LIN {X 0,Y 420.675,Z 239.811,A -85,B 0,C 180,E1 -10145.839,E2 -10145.839} C_VEL
LIN {X 0,Y 420.884,Z 242.407,A -85,B 0,C 180,E1 -10146.375,E2 -10146.375} C_VEL
LIN {X 0,Y 419.869,Z 259.45,A -85,B 0,C 180,E1 -10149.746,E2 -10149.746} C_VEL
LIN {X 0,Y 419.418,Z 267.017,A -85,B 0,C 180,E1 -10151.23,E2 -10151.23} C_VEL
LIN {X 0,Y 423.148,Z 292.501,A -85,B 0,C 180,E1 -10151.829,E2 -10151.829} C_VEL
LIN {X 0,Y 422.342,Z 375.452,A -85,B 0,C 180,E1 -10153.256,E2 -10153.256} C_VEL
LIN {X 0,Y 421.795,Z 388.688,A -85,B 0,C 180,E1 -10153.67,E2 -10153.67} C_VEL
LIN {X 0,Y 421.223,Z 401.426,A -85,B 0,C 180,E1 -10154.269,E2 -10154.269} C_VEL
LIN {X 0,Y 420.604,Z 412.728,A -85,B 0,C 180,E1 -10154.99,E2 -10154.99} C_VEL
LIN {X 0,Y 419.83,Z 424.418,A -85,B 0,C 180,E1 -10155.953,E2 -10155.953} C_VEL
LIN {X 0,Y 419.241,Z 434.93,A -85,B 0,C 180,E1 -10157.043,E2 -10157.043} C_VEL
LIN {X 0,Y 418.677,Z 443.516,A -85,B 0,C 180,E1 -10158.134,E2 -10158.134} C_VEL
LIN {X 0,Y 418.09,Z 451.424,A -85,B 0,C 180,E1 -10159.344,E2 -10159.344} C_VEL
LIN {X 0,Y 417.649,Z 459.143,A -85,B 0,C 180,E1 -10160.801,E2 -10160.801} C_VEL
LIN {X 0,Y 417.351,Z 465.34,A -85,B 0,C 180,E1 -10162.258,E2 -10162.258} C_VEL
LIN {X 0,Y 417.171,Z 470.222,A -85,B 0,C 180,E1 -10163.702,E2 -10163.702} C_VEL
LIN {X 0,Y 417.106,Z 474.036,A -85,B 0,C 180,E1 -10165.167,E2 -10165.167} C_VEL
LIN {X 0,Y 417.014,Z 475.982,A -85,B 0,C 180,E1 -10166.135,E2 -10166.135} C_VEL
LIN {X 0,Y 417.029,Z 477.511,A -85,B 0,C 180,E1 -10167.102,E2 -10167.102} C_VEL
LIN {X 0,Y 417.056,Z 478.586,A -85,B 0,C 180,E1 -10168.069,E2 -10168.069} C_VEL
LIN {X 0,Y 417.005,Z 479.55,A -85,B 0,C 180,E1 -10170,E2 -10170} C_VEL
LIN {X 0,Y 417.011,Z 479.453,A -85,B 0,C 180,E1 -10170.966,E2 -10170.966} C_VEL
LIN {X 0,Y 417.056,Z 478.925,A -85,B 0,C 180,E1 -10171.931,E2 -10171.931} C_VEL
LIN {X 0,Y 417.026,Z 477.997,A -85,B 0,C 180,E1 -10172.898,E2 -10172.898} C_VEL
LIN {X 0,Y 417.106,Z 474.952,A -85,B 0,C 180,E1 -10174.833,E2 -10174.833} C_VEL
LIN {X 0,Y 417.141,Z 471.563,A -85,B 0,C 180,E1 -10176.261,E2 -10176.261} C_VEL
LIN {X 0,Y 417.395,Z 466.962,A -85,B 0,C 180,E1 -10177.741,E2 -10177.741} C_VEL
LIN {X 0,Y 417.821,Z 460.107,A -85,B 0,C 180,E1 -10179.439,E2 -10179.439} C_VEL
LIN {X 0,Y 418.342,Z 452.686,A -85,B 0,C 180,E1 -10180.894,E2 -10180.894} C_VEL
LIN {X 0,Y 419.064,Z 445.134,A -85,B 0,C 180,E1 -10182.101,E2 -10182.101} C_VEL
LIN {X 0,Y 419.775,Z 436.004,A -85,B 0,C 180,E1 -10183.309,E2 -10183.309} C_VEL
LIN {X 0,Y 420.395,Z 426.465,A -85,B 0,C 180,E1 -10184.343,E2 -10184.343} C_VEL
LIN {X 0,Y 421.316,Z 414.675,A -85,B 0,C 180,E1 -10185.356,E2 -10185.356} C_VEL
LIN {X 0,Y 421.992,Z 404.07,A -85,B 0,C 180,E1 -10186.074,E2 -10186.074} C_VEL
LIN {X 0,Y 422.721,Z 391.294,A -85,B 0,C 180,E1 -10186.728,E2 -10186.728} C_VEL
LIN {X 0,Y 423.278,Z 378.466,A -85,B 0,C 180,E1 -10187.172,E2 -10187.172} C_VEL
LIN {X 0,Y 423.711,Z 360.488,A -85,B 0,C 180,E1 -10187.524,E2 -10187.524} C_VEL
LIN {X 0,Y 424.326,Z 291.938,A -85,B 0,C 180,E1 -10188.705,E2 -10188.705} C_VEL
LIN {X 0,Y 420.251,Z 268.65,A -85,B 0,C 180,E1 -10189.331,E2 -10189.331} C_VEL
LIN {X 0,Y 419.936,Z 266.884,A -85,B 0,C 180,E1 -10189.38,E2 -10189.38} C_VEL
LIN {X 0,Y 421.141,Z 249.854,A -85,B 0,C 180,E1 -10192.791,E2 -10192.791} C_VEL
LIN {X 0,Y 421.47,Z 243.375,A -85,B 0,C 180,E1 -10194.113,E2 -10194.113} C_VEL
LIN {X 0,Y 419.295,Z 232.058,A -85,B 0,C 180,E1 -10196.639,E2 -10196.639} C_VEL
LIN {X 0,Y 418.289,Z 227.385,A -85,B 0,C 180,E1 -10197.747,E2 -10197.747} C_VEL
LIN {X 0,Y 418.24,Z 227.389,A -85,B 0,C 180,E1 -10201.019,E2 -10201.019} C_VEL
LIN {X 0,Y 418.25,Z 227.388,A -85,B 0,C 180,E1 -10203.677,E2 -10203.677} C_VEL
LIN {X 0,Y 418.24,Z 227.389,A -85,B 0,C 180,E1 -10207.224,E2 -10207.224} C_VEL
LIN {X 0,Y 418.244,Z 227.389,A -85,B 0,C 180,E1 -10209.683,E2 -10209.683} C_VEL
LIN {X 0,Y 418.224,Z 227.387,A -85,B 0,C 180,E1 -10212.32,E2 -10212.32} C_VEL
LIN {X 0,Y 418.236,Z 227.388,A -85,B 0,C 180,E1 -10215.109,E2 -10215.109} C_VEL
LIN {X 0,Y 418.235,Z 227.389,A -85,B 0,C 180,E1 -10217.766,E2 -10217.766} C_VEL
LIN {X 0,Y 418.238,Z 227.389,A -85,B 0,C 180,E1 -10221.557,E2 -10221.557} C_VEL
LIN {X 0,Y 418.258,Z 227.385,A -85,B 0,C 180,E1 -10225.159,E2 -10225.159} C_VEL
LIN {X 0,Y 418.246,Z 227.385,A -85,B 0,C 180,E1 -10227.472,E2 -10227.472} C_VEL
LIN {X 0,Y 418.265,Z 227.377,A -85,B 0,C 180,E1 -10230.897,E2 -10230.897} C_VEL
LIN {X 0,Y 418.238,Z 227.38,A -85,B 0,C 180,E1 -10234.094,E2 -10234.094} C_VEL
LIN {X 0,Y 418.232,Z 227.39,A -85,B 0,C 180,E1 -10237.264,E2 -10237.264} C_VEL
LIN {X 0,Y 418.284,Z 227.378,A -85,B 0,C 180,E1 -10240.364,E2 -10240.364} C_VEL
LIN {X 0,Y 418.317,Z 227.374,A -85,B 0,C 180,E1 -10243.405,E2 -10243.405} C_VEL
LIN {X 0,Y 418.347,Z 227.372,A -85,B 0,C 180,E1 -10246.999,E2 -10246.999} C_VEL
LIN {X 0,Y 418.341,Z 227.371,A -85,B 0,C 180,E1 -10250.329,E2 -10250.329} C_VEL
LIN {X 0,Y 418.494,Z 227.35,A -85,B 0,C 180,E1 -10253.249,E2 -10253.249} C_VEL
LIN {X 0,Y 418.333,Z 227.375,A -85,B 0,C 180,E1 -10255.182,E2 -10255.182} C_VEL
LIN {X 0,Y 418.54,Z 227.342,A -85,B 0,C 180,E1 -10258.076,E2 -10258.076} C_VEL
LIN {X 0,Y 418.67,Z 227.331,A -85,B 0,C 180,E1 -10260,E2 -10260} C_VEL
LIN {X 0,Y 418.494,Z 227.35,A -85,B 0,C 180,E1 -10262.888,E2 -10262.888} C_VEL
LIN {X 0,Y 418.46,Z 227.356,A -85,B 0,C 180,E1 -10266.487,E2 -10266.487} C_VEL
LIN {X 0,Y 418.339,Z 227.376,A -85,B 0,C 180,E1 -10269.672,E2 -10269.672} C_VEL
LIN {X 0,Y 418.348,Z 227.37,A -85,B 0,C 180,E1 -10273.001,E2 -10273.001} C_VEL
LIN {X 0,Y 418.313,Z 227.374,A -85,B 0,C 180,E1 -10276.735,E2 -10276.735} C_VEL
LIN {X 0,Y 418.271,Z 227.382,A -85,B 0,C 180,E1 -10279.79,E2 -10279.79} C_VEL
LIN {X 0,Y 418.238,Z 227.378,A -85,B 0,C 180,E1 -10282.736,E2 -10282.736} C_VEL
LIN {X 0,Y 418.262,Z 227.378,A -85,B 0,C 180,E1 -10285.905,E2 -10285.905} C_VEL
LIN {X 0,Y 418.27,Z 227.384,A -85,B 0,C 180,E1 -10289.105,E2 -10289.105} C_VEL
LIN {X 0,Y 418.259,Z 227.383,A -85,B 0,C 180,E1 -10292.844,E2 -10292.844} C_VEL
LIN {X 0,Y 418.245,Z 227.381,A -85,B 0,C 180,E1 -10296.238,E2 -10296.238} C_VEL
LIN {X 0,Y 418.245,Z 227.388,A -85,B 0,C 180,E1 -10299.683,E2 -10299.683} C_VEL
LIN {X 0,Y 418.225,Z 227.387,A -85,B 0,C 180,E1 -10302.32,E2 -10302.32} C_VEL
LIN {X 0,Y 418.237,Z 227.39,A -85,B 0,C 180,E1 -10305.109,E2 -10305.109} C_VEL
LIN {X 0,Y 418.236,Z 227.391,A -85,B 0,C 180,E1 -10307.766,E2 -10307.766} C_VEL
LIN {X 0,Y 418.24,Z 227.394,A -85,B 0,C 180,E1 -10311.557,E2 -10311.557} C_VEL
LIN {X 0,Y 418.26,Z 227.389,A -85,B 0,C 180,E1 -10315.159,E2 -10315.159} C_VEL
LIN {X 0,Y 418.248,Z 227.388,A -85,B 0,C 180,E1 -10317.472,E2 -10317.472} C_VEL
LIN {X 0,Y 418.294,Z 227.523,A -85,B 0,C 180,E1 -10320.496,E2 -10320.496} C_VEL
LIN {X 0,Y 420.231,Z 237.183,A -85,B 0,C 180,E1 -10322.823,E2 -10322.823} C_VEL
LIN {X 0,Y 420.452,Z 242.272,A -85,B 0,C 180,E1 -10323.974,E2 -10323.974} C_VEL
LIN {X 0,Y 420.296,Z 245.419,A -85,B 0,C 180,E1 -10324.663,E2 -10324.663} C_VEL
LIN {X 0,Y 424.472,Z 264.589,A -85,B 0,C 180,E1 -10325.245,E2 -10325.245} C_VEL
LIN {X 0,Y 424.757,Z 269.362,A -85,B 0,C 180,E1 -10325.345,E2 -10325.345} C_VEL
LIN {X 0,Y 423.574,Z 353.087,A -85,B 0,C 180,E1 -10326.792,E2 -10326.792} C_VEL
LIN {X 0,Y 423.157,Z 366.435,A -85,B 0,C 180,E1 -10327.22,E2 -10327.22} C_VEL
LIN {X 0,Y 422.58,Z 379.229,A -85,B 0,C 180,E1 -10327.832,E2 -10327.832} C_VEL
LIN {X 0,Y 421.894,Z 390.948,A -85,B 0,C 180,E1 -10328.598,E2 -10328.598} C_VEL
LIN {X 0,Y 421.084,Z 402.881,A -85,B 0,C 180,E1 -10329.61,E2 -10329.61} C_VEL
LIN {X 0,Y 420.227,Z 413.237,A -85,B 0,C 180,E1 -10330.713,E2 -10330.713} C_VEL
LIN {X 0,Y 419.492,Z 422.499,A -85,B 0,C 180,E1 -10331.944,E2 -10331.944} C_VEL
LIN {X 0,Y 418.921,Z 429.828,A -85,B 0,C 180,E1 -10333.125,E2 -10333.125} C_VEL
LIN {X 0,Y 418.261,Z 437.559,A -85,B 0,C 180,E1 -10334.654,E2 -10334.654} C_VEL
LIN {X 0,Y 417.805,Z 444.366,A -85,B 0,C 180,E1 -10336.379,E2 -10336.379} C_VEL
LIN {X 0,Y 417.464,Z 449.019,A -85,B 0,C 180,E1 -10337.927,E2 -10337.927} C_VEL
LIN {X 0,Y 417.198,Z 452.2,A -85,B 0,C 180,E1 -10339.321,E2 -10339.321} C_VEL
LIN {X 0,Y 417.05,Z 454.001,A -85,B 0,C 180,E1 -10340.402,E2 -10340.402} C_VEL
LIN {X 0,Y 416.349,Z 455.082,A -85,B 0,C 180,E1 -10341.198,E2 -10341.198} C_VEL
LIN {X 0,Y 413.478,Z 456.229,A -85,B 0,C 180,E1 -10342.5,E2 -10342.5} C_VEL
LIN {X 0,Y 411.07,Z 456.634,A -85,B 0,C 180,E1 -10343.556,E2 -10343.556} C_VEL
LIN {X 0,Y 410.033,Z 456.603,A -85,B 0,C 180,E1 -10344.372,E2 -10344.372} C_VEL
LIN {X 0,Y 409.946,Z 456.468,A -85,B 0,C 180,E1 -10344.649,E2 -10344.649} C_VEL
LIN {X 0,Y 409.913,Z 455.619,A -85,B 0,C 180,E1 -10346.068,E2 -10346.068} C_VEL
LIN {X 0,Y 409.974,Z 454.491,A -85,B 0,C 180,E1 -10347.052,E2 -10347.052} C_VEL
LIN {X 0,Y 410.055,Z 452.937,A -85,B 0,C 180,E1 -10348.036,E2 -10348.036} C_VEL
LIN {X 0,Y 410.166,Z 449.828,A -85,B 0,C 180,E1 -10349.509,E2 -10349.509} C_VEL
LIN {X 0,Y 410.32,Z 445.675,A -85,B 0,C 180,E1 -10350.981,E2 -10350.981} C_VEL
LIN {X 0,Y 410.761,Z 439.351,A -85,B 0,C 180,E1 -10352.697,E2 -10352.697} C_VEL
LIN {X 0,Y 411.135,Z 432.478,A -85,B 0,C 180,E1 -10354.166,E2 -10354.166} C_VEL
LIN {X 0,Y 411.87,Z 423.849,A -85,B 0,C 180,E1 -10355.631,E2 -10355.631} C_VEL
LIN {X 0,Y 412.563,Z 415.025,A -85,B 0,C 180,E1 -10356.848,E2 -10356.848} C_VEL
LIN {X 0,Y 413.211,Z 405.345,A -85,B 0,C 180,E1 -10357.943,E2 -10357.943} C_VEL
LIN {X 0,Y 413.883,Z 394.726,A -85,B 0,C 180,E1 -10358.914,E2 -10358.914} C_VEL
LIN {X 0,Y 414.541,Z 382.831,A -85,B 0,C 180,E1 -10359.761,E2 -10359.761} C_VEL
LIN {X 0,Y 415.116,Z 370.445,A -85,B 0,C 180,E1 -10360.425,E2 -10360.425} C_VEL
LIN {X 0,Y 415.446,Z 357.479,A -85,B 0,C 180,E1 -10360.912,E2 -10360.912} C_VEL
LIN {X 0,Y 415.769,Z 341.674,A -85,B 0,C 180,E1 -10361.246,E2 -10361.246} C_VEL
LIN {X 0,Y 416.563,Z 266.126,A -85,B 0,C 180,E1 -10362.546,E2 -10362.546} C_VEL
LIN {X 0,Y 412.835,Z 245.467,A -85,B 0,C 180,E1 -10363.099,E2 -10363.099} C_VEL
LIN {X 0,Y 413.033,Z 237.818,A -85,B 0,C 180,E1 -10364.787,E2 -10364.787} C_VEL
LIN {X 0,Y 411.275,Z 228.258,A -85,B 0,C 180,E1 -10367.055,E2 -10367.055} C_VEL
LIN {X 0,Y 411.234,Z 228.257,A -85,B 0,C 180,E1 -10369.987,E2 -10369.987} C_VEL
LIN {X 0,Y 411.199,Z 228.262,A -85,B 0,C 180,E1 -10373.148,E2 -10373.148} C_VEL
LIN {X 0,Y 411.206,Z 228.263,A -85,B 0,C 180,E1 -10376.383,E2 -10376.383} C_VEL
LIN {X 0,Y 411.2,Z 228.26,A -85,B 0,C 180,E1 -10379.713,E2 -10379.713} C_VEL
LIN {X 0,Y 411.209,Z 228.261,A -85,B 0,C 180,E1 -10383.156,E2 -10383.156} C_VEL
LIN {X 0,Y 411.194,Z 228.266,A -85,B 0,C 180,E1 -10386.552,E2 -10386.552} C_VEL
LIN {X 0,Y 411.213,Z 228.258,A -85,B 0,C 180,E1 -10389.727,E2 -10389.727} C_VEL
LIN {X 0,Y 411.175,Z 228.265,A -85,B 0,C 180,E1 -10393.133,E2 -10393.133} C_VEL
LIN {X 0,Y 411.169,Z 228.264,A -85,B 0,C 180,E1 -10395.881,E2 -10395.881} C_VEL
LIN {X 0,Y 411.162,Z 228.271,A -85,B 0,C 180,E1 -10398.772,E2 -10398.772} C_VEL
LIN {X 0,Y 411.193,Z 228.262,A -85,B 0,C 180,E1 -10402.026,E2 -10402.026} C_VEL
LIN {X 0,Y 411.207,Z 228.259,A -85,B 0,C 180,E1 -10405.666,E2 -10405.666} C_VEL
LIN {X 0,Y 411.191,Z 228.263,A -85,B 0,C 180,E1 -10409.152,E2 -10409.152} C_VEL
LIN {X 0,Y 411.259,Z 228.258,A -85,B 0,C 180,E1 -10412.522,E2 -10412.522} C_VEL
LIN {X 0,Y 411.218,Z 228.258,A -85,B 0,C 180,E1 -10415.784,E2 -10415.784} C_VEL
LIN {X 0,Y 411.197,Z 228.264,A -85,B 0,C 180,E1 -10418.966,E2 -10418.966} C_VEL
LIN {X 0,Y 411.246,Z 228.256,A -85,B 0,C 180,E1 -10422.084,E2 -10422.084} C_VEL
LIN {X 0,Y 411.259,Z 228.254,A -85,B 0,C 180,E1 -10425.147,E2 -10425.147} C_VEL
LIN {X 0,Y 411.284,Z 228.252,A -85,B 0,C 180,E1 -10428.167,E2 -10428.167} C_VEL
LIN {X 0,Y 411.319,Z 228.247,A -85,B 0,C 180,E1 -10431.154,E2 -10431.154} C_VEL
LIN {X 0,Y 411.444,Z 228.231,A -85,B 0,C 180,E1 -10434.117,E2 -10434.117} C_VEL
LIN {X 0,Y 411.512,Z 228.222,A -85,B 0,C 180,E1 -10438.042,E2 -10438.042} C_VEL
LIN {X 0,Y 411.639,Z 228.206,A -85,B 0,C 180,E1 -10440,E2 -10440} C_VEL
LIN {X 0,Y 411.45,Z 228.232,A -85,B 0,C 180,E1 -10442.937,E2 -10442.937} C_VEL
LIN {X 0,Y 411.461,Z 228.231,A -85,B 0,C 180,E1 -10446.867,E2 -10446.867} C_VEL
LIN {X 0,Y 411.354,Z 228.245,A -85,B 0,C 180,E1 -10448.845,E2 -10448.845} C_VEL
LIN {X 0,Y 411.284,Z 228.25,A -85,B 0,C 180,E1 -10451.833,E2 -10451.833} C_VEL
LIN {X 0,Y 411.261,Z 228.256,A -85,B 0,C 180,E1 -10454.853,E2 -10454.853} C_VEL
LIN {X 0,Y 411.246,Z 228.255,A -85,B 0,C 180,E1 -10457.915,E2 -10457.915} C_VEL
LIN {X 0,Y 411.197,Z 228.263,A -85,B 0,C 180,E1 -10461.034,E2 -10461.034} C_VEL
LIN {X 0,Y 411.212,Z 228.261,A -85,B 0,C 180,E1 -10464.216,E2 -10464.216} C_VEL
LIN {X 0,Y 411.19,Z 228.261,A -85,B 0,C 180,E1 -10467.483,E2 -10467.483} C_VEL
LIN {X 0,Y 411.189,Z 228.265,A -85,B 0,C 180,E1 -10470.848,E2 -10470.848} C_VEL
LIN {X 0,Y 411.205,Z 228.264,A -85,B 0,C 180,E1 -10474.334,E2 -10474.334} C_VEL
LIN {X 0,Y 411.186,Z 228.263,A -85,B 0,C 180,E1 -10477.975,E2 -10477.975} C_VEL
LIN {X 0,Y 411.158,Z 228.266,A -85,B 0,C 180,E1 -10481.227,E2 -10481.227} C_VEL
LIN {X 0,Y 411.176,Z 228.27,A -85,B 0,C 180,E1 -10484.491,E2 -10484.491} C_VEL
LIN {X 0,Y 411.173,Z 228.266,A -85,B 0,C 180,E1 -10488.194,E2 -10488.194} C_VEL
LIN {X 0,Y 411.211,Z 228.263,A -85,B 0,C 180,E1 -10490.775,E2 -10490.775} C_VEL
LIN {X 0,Y 411.198,Z 228.267,A -85,B 0,C 180,E1 -10494.471,E2 -10494.471} C_VEL
LIN {X 0,Y 411.208,Z 228.262,A -85,B 0,C 180,E1 -10496.873,E2 -10496.873} C_VEL
LIN {X 0,Y 411.234,Z 228.262,A -85,B 0,C 180,E1 -10500.644,E2 -10500.644} C_VEL
LIN {X 0,Y 411.267,Z 228.273,A -85,B 0,C 180,E1 -10502.938,E2 -10502.938} C_VEL
LIN {X 0,Y 413.851,Z 242.011,A -85,B 0,C 180,E1 -10505.948,E2 -10505.948} C_VEL
LIN {X 0,Y 413.184,Z 254.87,A -85,B 0,C 180,E1 -10508.549,E2 -10508.549} C_VEL
LIN {X 0,Y 412.444,Z 266.837,A -85,B 0,C 180,E1 -10510.94,E2 -10510.94} C_VEL
LIN {X 0,Y 416.336,Z 293.443,A -85,B 0,C 180,E1 -10511.575,E2 -10511.575} C_VEL
LIN {X 0,Y 415.493,Z 375.167,A -85,B 0,C 180,E1 -10513.004,E2 -10513.004} C_VEL
LIN {X 0,Y 414.919,Z 388.433,A -85,B 0,C 180,E1 -10513.423,E2 -10513.423} C_VEL
LIN {X 0,Y 414.342,Z 400.618,A -85,B 0,C 180,E1 -10514,E2 -10514} C_VEL
LIN {X 0,Y 413.695,Z 412.093,A -85,B 0,C 180,E1 -10514.733,E2 -10514.733} C_VEL
LIN {X 0,Y 412.974,Z 422.96,A -85,B 0,C 180,E1 -10515.626,E2 -10515.626} C_VEL
LIN {X 0,Y 412.352,Z 433.674,A -85,B 0,C 180,E1 -10516.733,E2 -10516.733} C_VEL
LIN {X 0,Y 411.696,Z 443.084,A -85,B 0,C 180,E1 -10517.929,E2 -10517.929} C_VEL
LIN {X 0,Y 411.074,Z 451.034,A -85,B 0,C 180,E1 -10519.16,E2 -10519.16} C_VEL
LIN {X 0,Y 410.611,Z 458.8,A -85,B 0,C 180,E1 -10520.642,E2 -10520.642} C_VEL
LIN {X 0,Y 410.285,Z 465.025,A -85,B 0,C 180,E1 -10522.124,E2 -10522.124} C_VEL
LIN {X 0,Y 410.089,Z 470.291,A -85,B 0,C 180,E1 -10523.716,E2 -10523.716} C_VEL
LIN {X 0,Y 410.018,Z 473.771,A -85,B 0,C 180,E1 -10525.084,E2 -10525.084} C_VEL
LIN {X 0,Y 409.932,Z 475.729,A -85,B 0,C 180,E1 -10526.068,E2 -10526.068} C_VEL
LIN {X 0,Y 409.928,Z 477.272,A -85,B 0,C 180,E1 -10527.052,E2 -10527.052} C_VEL
LIN {X 0,Y 409.967,Z 478.364,A -85,B 0,C 180,E1 -10528.035,E2 -10528.035} C_VEL
LIN {X 0,Y 409.927,Z 479.349,A -85,B 0,C 180,E1 -10530,E2 -10530} C_VEL
LIN {X 0,Y 409.935,Z 479.264,A -85,B 0,C 180,E1 -10530.982,E2 -10530.982} C_VEL
LIN {X 0,Y 409.966,Z 478.754,A -85,B 0,C 180,E1 -10531.965,E2 -10531.965} C_VEL
LIN {X 0,Y 409.931,Z 476.527,A -85,B 0,C 180,E1 -10533.932,E2 -10533.932} C_VEL
LIN {X 0,Y 410.018,Z 473.761,A -85,B 0,C 180,E1 -10535.41,E2 -10535.41} C_VEL
LIN {X 0,Y 410.168,Z 469.98,A -85,B 0,C 180,E1 -10536.889,E2 -10536.889} C_VEL
LIN {X 0,Y 410.458,Z 465.087,A -85,B 0,C 180,E1 -10538.369,E2 -10538.369} C_VEL
LIN {X 0,Y 410.873,Z 458.938,A -85,B 0,C 180,E1 -10539.849,E2 -10539.849} C_VEL
LIN {X 0,Y 411.483,Z 451.303,A -85,B 0,C 180,E1 -10541.328,E2 -10541.328} C_VEL
LIN {X 0,Y 412.391,Z 441.724,A -85,B 0,C 180,E1 -10542.8,E2 -10542.8} C_VEL
LIN {X 0,Y 413.198,Z 431.201,A -85,B 0,C 180,E1 -10544.103,E2 -10544.103} C_VEL
LIN {X 0,Y 414.011,Z 420.791,A -85,B 0,C 180,E1 -10545.129,E2 -10545.129} C_VEL
LIN {X 0,Y 414.83,Z 409.964,A -85,B 0,C 180,E1 -10545.98,E2 -10545.98} C_VEL
LIN {X 0,Y 415.685,Z 398.027,A -85,B 0,C 180,E1 -10546.704,E2 -10546.704} C_VEL
LIN {X 0,Y 416.306,Z 386.64,A -85,B 0,C 180,E1 -10547.215,E2 -10547.215} C_VEL
LIN {X 0,Y 416.777,Z 373.651,A -85,B 0,C 180,E1 -10547.606,E2 -10547.606} C_VEL
LIN {X 0,Y 417.669,Z 292.562,A -85,B 0,C 180,E1 -10549.035,E2 -10549.035} C_VEL
LIN {X 0,Y 413.419,Z 268.529,A -85,B 0,C 180,E1 -10549.699,E2 -10549.699} C_VEL
LIN {X 0,Y 413.062,Z 266.681,A -85,B 0,C 180,E1 -10549.753,E2 -10549.753} C_VEL
LIN {X 0,Y 414.247,Z 250.906,A -85,B 0,C 180,E1 -10552.968,E2 -10552.968} C_VEL
LIN {X 0,Y 414.561,Z 244.622,A -85,B 0,C 180,E1 -10554.274,E2 -10554.274} C_VEL
LIN {X 0,Y 412.337,Z 233.31,A -85,B 0,C 180,E1 -10556.851,E2 -10556.851} C_VEL
LIN {X 0,Y 411.237,Z 228.263,A -85,B 0,C 180,E1 -10558.067,E2 -10558.067} C_VEL
LIN {X 0,Y 411.184,Z 228.268,A -85,B 0,C 180,E1 -10561.284,E2 -10561.284} C_VEL
LIN {X 0,Y 411.207,Z 228.261,A -85,B 0,C 180,E1 -10564.333,E2 -10564.333} C_VEL
LIN {X 0,Y 411.192,Z 228.265,A -85,B 0,C 180,E1 -10567.974,E2 -10567.974} C_VEL
LIN {X 0,Y 411.161,Z 228.271,A -85,B 0,C 180,E1 -10571.228,E2 -10571.228} C_VEL
LIN {X 0,Y 411.176,Z 228.265,A -85,B 0,C 180,E1 -10574.49,E2 -10574.49} C_VEL
LIN {X 0,Y 411.173,Z 228.265,A -85,B 0,C 180,E1 -10578.194,E2 -10578.194} C_VEL
LIN {X 0,Y 411.195,Z 228.263,A -85,B 0,C 180,E1 -10581.833,E2 -10581.833} C_VEL
LIN {X 0,Y 411.21,Z 228.263,A -85,B 0,C 180,E1 -10585.122,E2 -10585.122} C_VEL
LIN {X 0,Y 411.166,Z 228.266,A -85,B 0,C 180,E1 -10588.003,E2 -10588.003} C_VEL
LIN {X 0,Y 411.202,Z 228.262,A -85,B 0,C 180,E1 -10591.409,E2 -10591.409} C_VEL
LIN {X 0,Y 411.227,Z 228.254,A -85,B 0,C 180,E1 -10594.929,E2 -10594.929} C_VEL
LIN {X 0,Y 411.205,Z 228.259,A -85,B 0,C 180,E1 -10597.913,E2 -10597.913} C_VEL
LIN {X 0,Y 411.22,Z 228.261,A -85,B 0,C 180,E1 -10601.051,E2 -10601.051} C_VEL
LIN {X 0,Y 411.256,Z 228.253,A -85,B 0,C 180,E1 -10604.132,E2 -10604.132} C_VEL
LIN {X 0,Y 411.305,Z 228.251,A -85,B 0,C 180,E1 -10607.166,E2 -10607.166} C_VEL
LIN {X 0,Y 411.293,Z 228.249,A -85,B 0,C 180,E1 -10610.161,E2 -10610.161} C_VEL
LIN {X 0,Y 411.457,Z 228.226,A -85,B 0,C 180,E1 -10613.133,E2 -10613.133} C_VEL
LIN {X 0,Y 411.305,Z 228.249,A -85,B 0,C 180,E1 -10615.099,E2 -10615.099} C_VEL
LIN {X 0,Y 411.509,Z 228.217,A -85,B 0,C 180,E1 -10618.043,E2 -10618.043} C_VEL
LIN {X 0,Y 411.639,Z 228.207,A -85,B 0,C 180,E1 -10620,E2 -10620} C_VEL
LIN {X 0,Y 411.451,Z 228.227,A -85,B 0,C 180,E1 -10622.937,E2 -10622.937} C_VEL
LIN {X 0,Y 411.425,Z 228.234,A -85,B 0,C 180,E1 -10626.868,E2 -10626.868} C_VEL
LIN {X 0,Y 411.292,Z 228.252,A -85,B 0,C 180,E1 -10629.839,E2 -10629.839} C_VEL
LIN {X 0,Y 411.307,Z 228.247,A -85,B 0,C 180,E1 -10633.104,E2 -10633.104} C_VEL
LIN {X 0,Y 411.258,Z 228.254,A -85,B 0,C 180,E1 -10636.889,E2 -10636.889} C_VEL
LIN {X 0,Y 411.232,Z 228.257,A -85,B 0,C 180,E1 -10639.987,E2 -10639.987} C_VEL
LIN {X 0,Y 411.203,Z 228.258,A -85,B 0,C 180,E1 -10643.148,E2 -10643.148} C_VEL
LIN {X 0,Y 411.235,Z 228.251,A -85,B 0,C 180,E1 -10646.381,E2 -10646.381} C_VEL
LIN {X 0,Y 411.202,Z 228.261,A -85,B 0,C 180,E1 -10649.713,E2 -10649.713} C_VEL
LIN {X 0,Y 411.208,Z 228.263,A -85,B 0,C 180,E1 -10653.156,E2 -10653.156} C_VEL
LIN {X 0,Y 411.193,Z 228.259,A -85,B 0,C 180,E1 -10656.553,E2 -10656.553} C_VEL
LIN {X 0,Y 411.21,Z 228.264,A -85,B 0,C 180,E1 -10659.727,E2 -10659.727} C_VEL
LIN {X 0,Y 411.172,Z 228.27,A -85,B 0,C 180,E1 -10663.134,E2 -10663.134} C_VEL
LIN {X 0,Y 411.169,Z 228.264,A -85,B 0,C 180,E1 -10665.881,E2 -10665.881} C_VEL
LIN {X 0,Y 411.16,Z 228.272,A -85,B 0,C 180,E1 -10668.773,E2 -10668.773} C_VEL
LIN {X 0,Y 411.189,Z 228.268,A -85,B 0,C 180,E1 -10672.026,E2 -10672.026} C_VEL
LIN {X 0,Y 411.207,Z 228.266,A -85,B 0,C 180,E1 -10675.667,E2 -10675.667} C_VEL
LIN {X 0,Y 411.193,Z 228.263,A -85,B 0,C 180,E1 -10679.153,E2 -10679.153} C_VEL
LIN {X 0,Y 411.264,Z 228.376,A -85,B 0,C 180,E1 -10680.187,E2 -10680.187} C_VEL
LIN {X 0,Y 413.314,Z 238.501,A -85,B 0,C 180,E1 -10682.67,E2 -10682.67} C_VEL
LIN {X 0,Y 413.571,Z 243.31,A -85,B 0,C 180,E1 -10683.779,E2 -10683.779} C_VEL
LIN {X 0,Y 413.498,Z 245.961,A -85,B 0,C 180,E1 -10684.32,E2 -10684.32} C_VEL
LIN {X 0,Y 417.961,Z 266.179,A -85,B 0,C 180,E1 -10684.932,E2 -10684.932} C_VEL
LIN {X 0,Y 417.909,Z 285.188,A -85,B 0,C 180,E1 -10685.273,E2 -10685.273} C_VEL
LIN {X 0,Y 416.899,Z 352.988,A -85,B 0,C 180,E1 -10686.464,E2 -10686.464} C_VEL
LIN {X 0,Y 416.449,Z 366.429,A -85,B 0,C 180,E1 -10686.898,E2 -10686.898} C_VEL
LIN {X 0,Y 415.858,Z 379.279,A -85,B 0,C 180,E1 -10687.52,E2 -10687.52} C_VEL
LIN {X 0,Y 415.089,Z 391.579,A -85,B 0,C 180,E1 -10688.339,E2 -10688.339} C_VEL
LIN {X 0,Y 414.223,Z 403.641,A -85,B 0,C 180,E1 -10689.387,E2 -10689.387} C_VEL
LIN {X 0,Y 413.411,Z 412.832,A -85,B 0,C 180,E1 -10690.382,E2 -10690.382} C_VEL
LIN {X 0,Y 412.645,Z 422.227,A -85,B 0,C 180,E1 -10691.634,E2 -10691.634} C_VEL
LIN {X 0,Y 411.829,Z 431.287,A -85,B 0,C 180,E1 -10693.135,E2 -10693.135} C_VEL
LIN {X 0,Y 411.199,Z 438.557,A -85,B 0,C 180,E1 -10694.638,E2 -10694.638} C_VEL
LIN {X 0,Y 410.798,Z 444.329,A -85,B 0,C 180,E1 -10696.142,E2 -10696.142} C_VEL
LIN {X 0,Y 410.444,Z 448.263,A -85,B 0,C 180,E1 -10697.425,E2 -10697.425} C_VEL
LIN {X 0,Y 410.152,Z 452.268,A -85,B 0,C 180,E1 -10699.136,E2 -10699.136} C_VEL
LIN {X 0,Y 409.938,Z 455.243,A -85,B 0,C 180,E1 -10701.124,E2 -10701.124} C_VEL
LIN {X 0,Y 409.946,Z 456.131,A -85,B 0,C 180,E1 -10702.117,E2 -10702.117} C_VEL
LIN {X 0,Y 409.99,Z 456.691,A -85,B 0,C 180,E1 -10703.845,E2 -10703.845} C_VEL
LIN {X 0,Y 409.946,Z 456.468,A -85,B 0,C 180,E1 -10704.649,E2 -10704.649} C_VEL
LIN {X 0,Y 409.271,Z 456.126,A -85,B 0,C 180,E1 -10705.466,E2 -10705.466} C_VEL
LIN {X 0,Y 406.423,Z 454.934,A -85,B 0,C 180,E1 -10706.788,E2 -10706.788} C_VEL
LIN {X 0,Y 404.044,Z 453.498,A -85,B 0,C 180,E1 -10707.845,E2 -10707.845} C_VEL
LIN {X 0,Y 403.059,Z 452.059,A -85,B 0,C 180,E1 -10708.653,E2 -10708.653} C_VEL
LIN {X 0,Y 402.997,Z 451.472,A -85,B 0,C 180,E1 -10708.925,E2 -10708.925} C_VEL
LIN {X 0,Y 403.183,Z 447.579,A -85,B 0,C 180,E1 -10710.499,E2 -10710.499} C_VEL
LIN {X 0,Y 403.451,Z 442.723,A -85,B 0,C 180,E1 -10711.997,E2 -10711.997} C_VEL
LIN {X 0,Y 403.874,Z 436.611,A -85,B 0,C 180,E1 -10713.492,E2 -10713.492} C_VEL
LIN {X 0,Y 404.471,Z 429.012,A -85,B 0,C 180,E1 -10714.984,E2 -10714.984} C_VEL
LIN {X 0,Y 405.251,Z 419.467,A -85,B 0,C 180,E1 -10716.472,E2 -10716.472} C_VEL
LIN {X 0,Y 405.99,Z 409.633,A -85,B 0,C 180,E1 -10717.71,E2 -10717.71} C_VEL
LIN {X 0,Y 406.751,Z 398.56,A -85,B 0,C 180,E1 -10718.821,E2 -10718.821} C_VEL
LIN {X 0,Y 407.516,Z 385.976,A -85,B 0,C 180,E1 -10719.805,E2 -10719.805} C_VEL
LIN {X 0,Y 408.119,Z 374.629,A -85,B 0,C 180,E1 -10720.48,E2 -10720.48} C_VEL
LIN {X 0,Y 408.555,Z 361.103,A -85,B 0,C 180,E1 -10721.053,E2 -10721.053} C_VEL
LIN {X 0,Y 408.824,Z 348.21,A -85,B 0,C 180,E1 -10721.395,E2 -10721.395} C_VEL
LIN {X 0,Y 409.822,Z 267.593,A -85,B 0,C 180,E1 -10722.803,E2 -10722.803} C_VEL
LIN {X 0,Y 405.869,Z 245.693,A -85,B 0,C 180,E1 -10723.391,E2 -10723.391} C_VEL
LIN {X 0,Y 405.998,Z 238.317,A -85,B 0,C 180,E1 -10725.05,E2 -10725.05} C_VEL
LIN {X 0,Y 404.227,Z 229.136,A -85,B 0,C 180,E1 -10727.257,E2 -10727.257} C_VEL
LIN {X 0,Y 404.167,Z 229.139,A -85,B 0,C 180,E1 -10730.351,E2 -10730.351} C_VEL
LIN {X 0,Y 404.163,Z 229.137,A -85,B 0,C 180,E1 -10733.575,E2 -10733.575} C_VEL
LIN {X 0,Y 404.154,Z 229.143,A -85,B 0,C 180,E1 -10736.88,E2 -10736.88} C_VEL
LIN {X 0,Y 404.147,Z 229.141,A -85,B 0,C 180,E1 -10740.285,E2 -10740.285} C_VEL
LIN {X 0,Y 404.147,Z 229.139,A -85,B 0,C 180,E1 -10743.812,E2 -10743.812} C_VEL
LIN {X 0,Y 404.138,Z 229.144,A -85,B 0,C 180,E1 -10746.875,E2 -10746.875} C_VEL
LIN {X 0,Y 404.149,Z 229.139,A -85,B 0,C 180,E1 -10750.08,E2 -10750.08} C_VEL
LIN {X 0,Y 404.154,Z 229.14,A -85,B 0,C 180,E1 -10753.083,E2 -10753.083} C_VEL
LIN {X 0,Y 404.149,Z 229.139,A -85,B 0,C 180,E1 -10755.926,E2 -10755.926} C_VEL
LIN {X 0,Y 404.117,Z 229.149,A -85,B 0,C 180,E1 -10758.634,E2 -10758.634} C_VEL
LIN {X 0,Y 404.151,Z 229.138,A -85,B 0,C 180,E1 -10761.493,E2 -10761.493} C_VEL
LIN {X 0,Y 404.185,Z 229.137,A -85,B 0,C 180,E1 -10764.984,E2 -10764.984} C_VEL
LIN {X 0,Y 404.144,Z 229.145,A -85,B 0,C 180,E1 -10768.554,E2 -10768.554} C_VEL
LIN {X 0,Y 404.196,Z 229.133,A -85,B 0,C 180,E1 -10772,E2 -10772} C_VEL
LIN {X 0,Y 404.173,Z 229.136,A -85,B 0,C 180,E1 -10775.334,E2 -10775.334} C_VEL
LIN {X 0,Y 404.161,Z 229.144,A -85,B 0,C 180,E1 -10778.582,E2 -10778.582} C_VEL
LIN {X 0,Y 404.205,Z 229.131,A -85,B 0,C 180,E1 -10781.762,E2 -10781.762} C_VEL
LIN {X 0,Y 404.206,Z 229.135,A -85,B 0,C 180,E1 -10784.882,E2 -10784.882} C_VEL
LIN {X 0,Y 404.257,Z 229.126,A -85,B 0,C 180,E1 -10787.958,E2 -10787.958} C_VEL
LIN {X 0,Y 404.266,Z 229.127,A -85,B 0,C 180,E1 -10790.998,E2 -10790.998} C_VEL
LIN {X 0,Y 404.394,Z 229.109,A -85,B 0,C 180,E1 -10794.014,E2 -10794.014} C_VEL
LIN {X 0,Y 404.481,Z 229.098,A -85,B 0,C 180,E1 -10798.008,E2 -10798.008} C_VEL
LIN {X 0,Y 404.608,Z 229.082,A -85,B 0,C 180,E1 -10800,E2 -10800} C_VEL
LIN {X 0,Y 404.409,Z 229.109,A -85,B 0,C 180,E1 -10802.988,E2 -10802.988} C_VEL
LIN {X 0,Y 404.412,Z 229.108,A -85,B 0,C 180,E1 -10806.987,E2 -10806.987} C_VEL
LIN {X 0,Y 404.258,Z 229.126,A -85,B 0,C 180,E1 -10810.012,E2 -10810.012} C_VEL
LIN {X 0,Y 404.267,Z 229.125,A -85,B 0,C 180,E1 -10813.211,E2 -10813.211} C_VEL
LIN {X 0,Y 404.216,Z 229.132,A -85,B 0,C 180,E1 -10817.007,E2 -10817.007} C_VEL
LIN {X 0,Y 404.164,Z 229.141,A -85,B 0,C 180,E1 -10820.352,E2 -10820.352} C_VEL
LIN {X 0,Y 404.161,Z 229.137,A -85,B 0,C 180,E1 -10823.575,E2 -10823.575} C_VEL
LIN {X 0,Y 404.136,Z 229.144,A -85,B 0,C 180,E1 -10826.881,E2 -10826.881} C_VEL
LIN {X 0,Y 404.145,Z 229.143,A -85,B 0,C 180,E1 -10830.285,E2 -10830.285} C_VEL
LIN {X 0,Y 404.144,Z 229.139,A -85,B 0,C 180,E1 -10833.812,E2 -10833.812} C_VEL
LIN {X 0,Y 404.134,Z 229.144,A -85,B 0,C 180,E1 -10836.875,E2 -10836.875} C_VEL
LIN {X 0,Y 404.12,Z 229.144,A -85,B 0,C 180,E1 -10840.075,E2 -10840.075} C_VEL
LIN {X 0,Y 404.15,Z 229.14,A -85,B 0,C 180,E1 -10843.083,E2 -10843.083} C_VEL
LIN {X 0,Y 404.148,Z 229.139,A -85,B 0,C 180,E1 -10845.926,E2 -10845.926} C_VEL
LIN {X 0,Y 404.116,Z 229.149,A -85,B 0,C 180,E1 -10848.635,E2 -10848.635} C_VEL
LIN {X 0,Y 404.15,Z 229.138,A -85,B 0,C 180,E1 -10851.493,E2 -10851.493} C_VEL
LIN {X 0,Y 404.185,Z 229.136,A -85,B 0,C 180,E1 -10854.984,E2 -10854.984} C_VEL
LIN {X 0,Y 404.143,Z 229.146,A -85,B 0,C 180,E1 -10858.554,E2 -10858.554} C_VEL
LIN {X 0,Y 404.196,Z 229.138,A -85,B 0,C 180,E1 -10862,E2 -10862} C_VEL
LIN {X 0,Y 404.241,Z 229.148,A -85,B 0,C 180,E1 -10862.707,E2 -10862.707} C_VEL
LIN {X 0,Y 406.791,Z 242.684,A -85,B 0,C 180,E1 -10865.73,E2 -10865.73} C_VEL
LIN {X 0,Y 406.637,Z 249.347,A -85,B 0,C 180,E1 -10867.116,E2 -10867.116} C_VEL
LIN {X 0,Y 405.504,Z 266.643,A -85,B 0,C 180,E1 -10870.64,E2 -10870.64} C_VEL
LIN {X 0,Y 409.518,Z 294.222,A -85,B 0,C 180,E1 -10871.311,E2 -10871.311} C_VEL
LIN {X 0,Y 408.64,Z 374.849,A -85,B 0,C 180,E1 -10872.742,E2 -10872.742} C_VEL
LIN {X 0,Y 408.068,Z 388.159,A -85,B 0,C 180,E1 -10873.169,E2 -10873.169} C_VEL
LIN {X 0,Y 407.511,Z 399.799,A -85,B 0,C 180,E1 -10873.725,E2 -10873.725} C_VEL
LIN {X 0,Y 406.825,Z 411.426,A -85,B 0,C 180,E1 -10874.469,E2 -10874.469} C_VEL
LIN {X 0,Y 405.997,Z 423.319,A -85,B 0,C 180,E1 -10875.463,E2 -10875.463} C_VEL
LIN {X 0,Y 405.354,Z 433.69,A -85,B 0,C 180,E1 -10876.559,E2 -10876.559} C_VEL
LIN {X 0,Y 404.727,Z 442.645,A -85,B 0,C 180,E1 -10877.718,E2 -10877.718} C_VEL
LIN {X 0,Y 404.056,Z 450.635,A -85,B 0,C 180,E1 -10878.97,E2 -10878.97} C_VEL
LIN {X 0,Y 403.579,Z 458.453,A -85,B 0,C 180,E1 -10880.478,E2 -10880.478} C_VEL
LIN {X 0,Y 403.218,Z 464.706,A -85,B 0,C 180,E1 -10881.985,E2 -10881.985} C_VEL
LIN {X 0,Y 402.981,Z 470.458,A -85,B 0,C 180,E1 -10883.765,E2 -10883.765} C_VEL
LIN {X 0,Y 402.93,Z 473.503,A -85,B 0,C 180,E1 -10884.997,E2 -10884.997} C_VEL
LIN {X 0,Y 402.852,Z 475.473,A -85,B 0,C 180,E1 -10885.999,E2 -10885.999} C_VEL
LIN {X 0,Y 402.827,Z 477.029,A -85,B 0,C 180,E1 -10887,E2 -10887} C_VEL
LIN {X 0,Y 402.865,Z 478.141,A -85,B 0,C 180,E1 -10888.001,E2 -10888.001} C_VEL
LIN {X 0,Y 402.862,Z 478.838,A -85,B 0,C 180,E1 -10889,E2 -10889} C_VEL
LIN {X 0,Y 402.862,Z 479.074,A -85,B 0,C 180,E1 -10891,E2 -10891} C_VEL
LIN {X 0,Y 402.864,Z 478.583,A -85,B 0,C 180,E1 -10892,E2 -10892} C_VEL
LIN {X 0,Y 402.851,Z 476.378,A -85,B 0,C 180,E1 -10894.002,E2 -10894.002} C_VEL
LIN {X 0,Y 402.917,Z 473.634,A -85,B 0,C 180,E1 -10895.505,E2 -10895.505} C_VEL
LIN {X 0,Y 403.083,Z 469.877,A -85,B 0,C 180,E1 -10897.01,E2 -10897.01} C_VEL
LIN {X 0,Y 403.396,Z 465.011,A -85,B 0,C 180,E1 -10898.516,E2 -10898.516} C_VEL
LIN {X 0,Y 403.858,Z 458.891,A -85,B 0,C 180,E1 -10900.022,E2 -10900.022} C_VEL
LIN {X 0,Y 404.512,Z 451.297,A -85,B 0,C 180,E1 -10901.525,E2 -10901.525} C_VEL
LIN {X 0,Y 405.317,Z 443.542,A -85,B 0,C 180,E1 -10902.772,E2 -10902.772} C_VEL
LIN {X 0,Y 406.208,Z 433.102,A -85,B 0,C 180,E1 -10904.136,E2 -10904.136} C_VEL
LIN {X 0,Y 407.046,Z 422.333,A -85,B 0,C 180,E1 -10905.266,E2 -10905.266} C_VEL
LIN {X 0,Y 407.903,Z 411.986,A -85,B 0,C 180,E1 -10906.131,E2 -10906.131} C_VEL
LIN {X 0,Y 408.749,Z 400.708,A -85,B 0,C 180,E1 -10906.867,E2 -10906.867} C_VEL
LIN {X 0,Y 409.473,Z 388.051,A -85,B 0,C 180,E1 -10907.479,E2 -10907.479} C_VEL
LIN {X 0,Y 410.071,Z 374.894,A -85,B 0,C 180,E1 -10907.904,E2 -10907.904} C_VEL
LIN {X 0,Y 411.107,Z 293.773,A -85,B 0,C 180,E1 -10909.362,E2 -10909.362} C_VEL
LIN {X 0,Y 407.006,Z 270.514,A -85,B 0,C 180,E1 -10910.019,E2 -10910.019} C_VEL
LIN {X 0,Y 406.231,Z 266.32,A -85,B 0,C 180,E1 -10910.171,E2 -10910.171} C_VEL
LIN {X 0,Y 407.611,Z 248.783,A -85,B 0,C 180,E1 -10913.817,E2 -10913.817} C_VEL
LIN {X 0,Y 407.61,Z 245.869,A -85,B 0,C 180,E1 -10914.444,E2 -10914.444} C_VEL
LIN {X 0,Y 405.231,Z 233.876,A -85,B 0,C 180,E1 -10917.234,E2 -10917.234} C_VEL
LIN {X 0,Y 404.196,Z 229.141,A -85,B 0,C 180,E1 -10918.424,E2 -10918.424} C_VEL
LIN {X 0,Y 404.141,Z 229.144,A -85,B 0,C 180,E1 -10921.558,E2 -10921.558} C_VEL
LIN {X 0,Y 404.185,Z 229.136,A -85,B 0,C 180,E1 -10925.016,E2 -10925.016} C_VEL
LIN {X 0,Y 404.151,Z 229.141,A -85,B 0,C 180,E1 -10928.757,E2 -10928.757} C_VEL
LIN {X 0,Y 404.12,Z 229.148,A -85,B 0,C 180,E1 -10931.599,E2 -10931.599} C_VEL
LIN {X 0,Y 404.146,Z 229.14,A -85,B 0,C 180,E1 -10934.522,E2 -10934.522} C_VEL
LIN {X 0,Y 404.133,Z 229.147,A -85,B 0,C 180,E1 -10937.295,E2 -10937.295} C_VEL
LIN {X 0,Y 404.132,Z 229.143,A -85,B 0,C 180,E1 -10939.951,E2 -10939.951} C_VEL
LIN {X 0,Y 404.135,Z 229.141,A -85,B 0,C 180,E1 -10943.125,E2 -10943.125} C_VEL
LIN {X 0,Y 404.145,Z 229.136,A -85,B 0,C 180,E1 -10946.188,E2 -10946.188} C_VEL
LIN {X 0,Y 404.145,Z 229.138,A -85,B 0,C 180,E1 -10949.715,E2 -10949.715} C_VEL
LIN {X 0,Y 404.152,Z 229.142,A -85,B 0,C 180,E1 -10953.12,E2 -10953.12} C_VEL
LIN {X 0,Y 404.161,Z 229.138,A -85,B 0,C 180,E1 -10956.425,E2 -10956.425} C_VEL
LIN {X 0,Y 404.192,Z 229.136,A -85,B 0,C 180,E1 -10959.874,E2 -10959.874} C_VEL
LIN {X 0,Y 404.217,Z 229.131,A -85,B 0,C 180,E1 -10962.993,E2 -10962.993} C_VEL
LIN {X 0,Y 404.284,Z 229.123,A -85,B 0,C 180,E1 -10966.939,E2 -10966.939} C_VEL
LIN {X 0,Y 404.258,Z 229.127,A -85,B 0,C 180,E1 -10969.988,E2 -10969.988} C_VEL
LIN {X 0,Y 404.404,Z 229.104,A -85,B 0,C 180,E1 -10973.013,E2 -10973.013} C_VEL
LIN {X 0,Y 404.278,Z 229.124,A -85,B 0,C 180,E1 -10975.014,E2 -10975.014} C_VEL
LIN {X 0,Y 404.477,Z 229.093,A -85,B 0,C 180,E1 -10978.009,E2 -10978.009} C_VEL
LIN {X 0,Y 404.608,Z 229.083,A -85,B 0,C 180,E1 -10980,E2 -10980} C_VEL
LIN {X 0,Y 404.409,Z 229.105,A -85,B 0,C 180,E1 -10982.989,E2 -10982.989} C_VEL
LIN {X 0,Y 404.371,Z 229.113,A -85,B 0,C 180,E1 -10986.988,E2 -10986.988} C_VEL
LIN {X 0,Y 404.257,Z 229.127,A -85,B 0,C 180,E1 -10990.012,E2 -10990.012} C_VEL
LIN {X 0,Y 404.268,Z 229.123,A -85,B 0,C 180,E1 -10993.211,E2 -10993.211} C_VEL
LIN {X 0,Y 404.217,Z 229.132,A -85,B 0,C 180,E1 -10997.007,E2 -10997.007} C_VEL
LIN {X 0,Y 404.165,Z 229.136,A -85,B 0,C 180,E1 -11000.352,E2 -11000.352} C_VEL
LIN {X 0,Y 404.166,Z 229.14,A -85,B 0,C 180,E1 -11003.575,E2 -11003.575} C_VEL
LIN {X 0,Y 404.182,Z 229.133,A -85,B 0,C 180,E1 -11005.767,E2 -11005.767} C_VEL
LIN {X 0,Y 404.196,Z 229.134,A -85,B 0,C 180,E1 -11008,E2 -11008} C_VEL
LIN {X 0,Y 404.141,Z 229.146,A -85,B 0,C 180,E1 -11011.558,E2 -11011.558} C_VEL
LIN {X 0,Y 404.186,Z 229.138,A -85,B 0,C 180,E1 -11015.016,E2 -11015.016} C_VEL
LIN {X 0,Y 404.151,Z 229.14,A -85,B 0,C 180,E1 -11018.758,E2 -11018.758} C_VEL
LIN {X 0,Y 404.121,Z 229.147,A -85,B 0,C 180,E1 -11021.599,E2 -11021.599} C_VEL
LIN {X 0,Y 404.147,Z 229.142,A -85,B 0,C 180,E1 -11024.522,E2 -11024.522} C_VEL
LIN {X 0,Y 404.134,Z 229.141,A -85,B 0,C 180,E1 -11027.295,E2 -11027.295} C_VEL
LIN {X 0,Y 404.134,Z 229.142,A -85,B 0,C 180,E1 -11029.951,E2 -11029.951} C_VEL
LIN {X 0,Y 404.137,Z 229.15,A -85,B 0,C 180,E1 -11033.126,E2 -11033.126} C_VEL
LIN {X 0,Y 404.147,Z 229.143,A -85,B 0,C 180,E1 -11036.188,E2 -11036.188} C_VEL
LIN {X 0,Y 404.181,Z 229.199,A -85,B 0,C 180,E1 -11039.852,E2 -11039.852} C_VEL
LIN {X 0,Y 406.519,Z 240.743,A -85,B 0,C 180,E1 -11042.733,E2 -11042.733} C_VEL
LIN {X 0,Y 406.59,Z 245.787,A -85,B 0,C 180,E1 -11043.9,E2 -11043.9} C_VEL
LIN {X 0,Y 410.824,Z 264.542,A -85,B 0,C 180,E1 -11044.513,E2 -11044.513} C_VEL
LIN {X 0,Y 411.529,Z 269.329,A -85,B 0,C 180,E1 -11044.64,E2 -11044.64} C_VEL
LIN {X 0,Y 410.198,Z 354.073,A -85,B 0,C 180,E1 -11046.157,E2 -11046.157} C_VEL
LIN {X 0,Y 409.739,Z 367.22,A -85,B 0,C 180,E1 -11046.598,E2 -11046.598} C_VEL
LIN {X 0,Y 409.153,Z 379.342,A -85,B 0,C 180,E1 -11047.198,E2 -11047.198} C_VEL
LIN {X 0,Y 408.377,Z 391.216,A -85,B 0,C 180,E1 -11047.993,E2 -11047.993} C_VEL
LIN {X 0,Y 407.463,Z 403.102,A -85,B 0,C 180,E1 -11049.029,E2 -11049.029} C_VEL
LIN {X 0,Y 406.589,Z 412.419,A -85,B 0,C 180,E1 -11050.039,E2 -11050.039} C_VEL
LIN {X 0,Y 405.788,Z 421.959,A -85,B 0,C 180,E1 -11051.312,E2 -11051.312} C_VEL
LIN {X 0,Y 404.95,Z 431.099,A -85,B 0,C 180,E1 -11052.84,E2 -11052.84} C_VEL
LIN {X 0,Y 404.258,Z 438.436,A -85,B 0,C 180,E1 -11054.367,E2 -11054.367} C_VEL
LIN {X 0,Y 403.784,Z 444.284,A -85,B 0,C 180,E1 -11055.896,E2 -11055.896} C_VEL
LIN {X 0,Y 403.399,Z 448.606,A -85,B 0,C 180,E1 -11057.327,E2 -11057.327} C_VEL
LIN {X 0,Y 403.112,Z 452.329,A -85,B 0,C 180,E1 -11058.943,E2 -11058.943} C_VEL
LIN {X 0,Y 402.912,Z 454.053,A -85,B 0,C 180,E1 -11059.954,E2 -11059.954} C_VEL
LIN {X 0,Y 402.85,Z 456.272,A -85,B 0,C 180,E1 -11061.977,E2 -11061.977} C_VEL
LIN {X 0,Y 402.895,Z 456.877,A -85,B 0,C 180,E1 -11063.879,E2 -11063.879} C_VEL
LIN {X 0,Y 402.863,Z 456.556,A -85,B 0,C 180,E1 -11064.996,E2 -11064.996} C_VEL
LIN {X 0,Y 402.831,Z 455.872,A -85,B 0,C 180,E1 -11065.998,E2 -11065.998} C_VEL
LIN {X 0,Y 402.871,Z 454.789,A -85,B 0,C 180,E1 -11067,E2 -11067} C_VEL
LIN {X 0,Y 402.98,Z 453.259,A -85,B 0,C 180,E1 -11068.001,E2 -11068.001} C_VEL
LIN {X 0,Y 402.997,Z 451.472,A -85,B 0,C 180,E1 -11068.925,E2 -11068.925} C_VEL
LIN {X 0,Y 402.424,Z 449.762,A -85,B 0,C 180,E1 -11069.725,E2 -11069.725} C_VEL
LIN {X 0,Y 399.793,Z 446.38,A -85,B 0,C 180,E1 -11071.001,E2 -11071.001} C_VEL
LIN {X 0,Y 397.181,Z 442.333,A -85,B 0,C 180,E1 -11072.251,E2 -11072.251} C_VEL
LIN {X 0,Y 396.654,Z 439.486,A -85,B 0,C 180,E1 -11073.002,E2 -11073.002} C_VEL
LIN {X 0,Y 397.196,Z 432.29,A -85,B 0,C 180,E1 -11074.567,E2 -11074.567} C_VEL
LIN {X 0,Y 397.919,Z 423.538,A -85,B 0,C 180,E1 -11076.083,E2 -11076.083} C_VEL
LIN {X 0,Y 398.756,Z 413.594,A -85,B 0,C 180,E1 -11077.469,E2 -11077.469} C_VEL
LIN {X 0,Y 399.522,Z 403.431,A -85,B 0,C 180,E1 -11078.599,E2 -11078.599} C_VEL
LIN {X 0,Y 400.286,Z 392.171,A -85,B 0,C 180,E1 -11079.602,E2 -11079.602} C_VEL
LIN {X 0,Y 400.906,Z 380.503,A -85,B 0,C 180,E1 -11080.415,E2 -11080.415} C_VEL
LIN {X 0,Y 401.506,Z 368.423,A -85,B 0,C 180,E1 -11081.037,E2 -11081.037} C_VEL
LIN {X 0,Y 401.832,Z 354.667,A -85,B 0,C 180,E1 -11081.52,E2 -11081.52} C_VEL
LIN {X 0,Y 402.417,Z 318.49,A -85,B 0,C 180,E1 -11082.193,E2 -11082.193} C_VEL
LIN {X 0,Y 402.965,Z 267.983,A -85,B 0,C 180,E1 -11083.093,E2 -11083.093} C_VEL
LIN {X 0,Y 398.953,Z 245.976,A -85,B 0,C 180,E1 -11083.679,E2 -11083.679} C_VEL
LIN {X 0,Y 399.087,Z 240.055,A -85,B 0,C 180,E1 -11085.029,E2 -11085.029} C_VEL
LIN {X 0,Y 397.194,Z 230.011,A -85,B 0,C 180,E1 -11087.506,E2 -11087.506} C_VEL
LIN {X 0,Y 397.106,Z 230.023,A -85,B 0,C 180,E1 -11090.73,E2 -11090.73} C_VEL
LIN {X 0,Y 397.126,Z 230.014,A -85,B 0,C 180,E1 -11094.019,E2 -11094.019} C_VEL
LIN {X 0,Y 397.118,Z 230.014,A -85,B 0,C 180,E1 -11097.763,E2 -11097.763} C_VEL
LIN {X 0,Y 397.081,Z 230.024,A -85,B 0,C 180,E1 -11100.882,E2 -11100.882} C_VEL
LIN {X 0,Y 397.128,Z 230.018,A -85,B 0,C 180,E1 -11104.493,E2 -11104.493} C_VEL
LIN {X 0,Y 397.103,Z 230.019,A -85,B 0,C 180,E1 -11108.275,E2 -11108.275} C_VEL
LIN {X 0,Y 397.09,Z 230.022,A -85,B 0,C 180,E1 -11110.909,E2 -11110.909} C_VEL
LIN {X 0,Y 397.102,Z 230.016,A -85,B 0,C 180,E1 -11113.648,E2 -11113.648} C_VEL
LIN {X 0,Y 397.102,Z 230.022,A -85,B 0,C 180,E1 -11116.521,E2 -11116.521} C_VEL
LIN {X 0,Y 397.114,Z 230.019,A -85,B 0,C 180,E1 -11120.422,E2 -11120.422} C_VEL
LIN {X 0,Y 397.109,Z 230.018,A -85,B 0,C 180,E1 -11124.265,E2 -11124.265} C_VEL
LIN {X 0,Y 397.116,Z 230.021,A -85,B 0,C 180,E1 -11126.727,E2 -11126.727} C_VEL
LIN {X 0,Y 397.126,Z 230.016,A -85,B 0,C 180,E1 -11130.296,E2 -11130.296} C_VEL
LIN {X 0,Y 397.195,Z 230.012,A -85,B 0,C 180,E1 -11132.61,E2 -11132.61} C_VEL
LIN {X 0,Y 397.13,Z 230.014,A -85,B 0,C 180,E1 -11135.981,E2 -11135.981} C_VEL
LIN {X 0,Y 397.14,Z 230.011,A -85,B 0,C 180,E1 -11139.704,E2 -11139.704} C_VEL
LIN {X 0,Y 397.183,Z 230.011,A -85,B 0,C 180,E1 -11142.845,E2 -11142.845} C_VEL
LIN {X 0,Y 397.229,Z 230.007,A -85,B 0,C 180,E1 -11146.703,E2 -11146.703} C_VEL
LIN {X 0,Y 397.217,Z 230.002,A -85,B 0,C 180,E1 -11149.809,E2 -11149.809} C_VEL
LIN {X 0,Y 397.319,Z 229.993,A -85,B 0,C 180,E1 -11152.887,E2 -11152.887} C_VEL
LIN {X 0,Y 397.247,Z 230.002,A -85,B 0,C 180,E1 -11154.925,E2 -11154.925} C_VEL
LIN {X 0,Y 397.45,Z 229.974,A -85,B 0,C 180,E1 -11157.973,E2 -11157.973} C_VEL
LIN {X 0,Y 397.577,Z 229.958,A -85,B 0,C 180,E1 -11160,E2 -11160} C_VEL
LIN {X 0,Y 397.368,Z 229.985,A -85,B 0,C 180,E1 -11163.041,E2 -11163.041} C_VEL
LIN {X 0,Y 397.365,Z 229.985,A -85,B 0,C 180,E1 -11167.112,E2 -11167.112} C_VEL
LIN {X 0,Y 397.217,Z 230.004,A -85,B 0,C 180,E1 -11170.191,E2 -11170.191} C_VEL
LIN {X 0,Y 397.227,Z 230.001,A -85,B 0,C 180,E1 -11173.321,E2 -11173.321} C_VEL
LIN {X 0,Y 397.182,Z 230.007,A -85,B 0,C 180,E1 -11177.155,E2 -11177.155} C_VEL
LIN {X 0,Y 397.103,Z 230.021,A -85,B 0,C 180,E1 -11180.73,E2 -11180.73} C_VEL
LIN {X 0,Y 397.124,Z 230.015,A -85,B 0,C 180,E1 -11184.019,E2 -11184.019} C_VEL
LIN {X 0,Y 397.102,Z 230.016,A -85,B 0,C 180,E1 -11187.397,E2 -11187.397} C_VEL
LIN {X 0,Y 397.078,Z 230.023,A -85,B 0,C 180,E1 -11190.883,E2 -11190.883} C_VEL
LIN {X 0,Y 397.125,Z 230.02,A -85,B 0,C 180,E1 -11194.493,E2 -11194.493} C_VEL
LIN {X 0,Y 397.093,Z 230.021,A -85,B 0,C 180,E1 -11198.276,E2 -11198.276} C_VEL
LIN {X 0,Y 397.061,Z 230.023,A -85,B 0,C 180,E1 -11201.978,E2 -11201.978} C_VEL
LIN {X 0,Y 397.087,Z 230.02,A -85,B 0,C 180,E1 -11205.069,E2 -11205.069} C_VEL
LIN {X 0,Y 397.063,Z 230.023,A -85,B 0,C 180,E1 -11208.022,E2 -11208.022} C_VEL
LIN {X 0,Y 397.127,Z 230.014,A -85,B 0,C 180,E1 -11211.139,E2 -11211.139} C_VEL
LIN {X 0,Y 397.12,Z 230.021,A -85,B 0,C 180,E1 -11214.497,E2 -11214.497} C_VEL
LIN {X 0,Y 397.079,Z 230.02,A -85,B 0,C 180,E1 -11217.929,E2 -11217.929} C_VEL
LIN {X 0,Y 397.123,Z 230.017,A -85,B 0,C 180,E1 -11221.456,E2 -11221.456} C_VEL
LIN {X 0,Y 397.198,Z 230.024,A -85,B 0,C 180,E1 -11222.467,E2 -11222.467} C_VEL
LIN {X 0,Y 399.807,Z 243.791,A -85,B 0,C 180,E1 -11225.601,E2 -11225.601} C_VEL
LIN {X 0,Y 399.756,Z 248.953,A -85,B 0,C 180,E1 -11226.699,E2 -11226.699} C_VEL
LIN {X 0,Y 398.577,Z 266.428,A -85,B 0,C 180,E1 -11230.326,E2 -11230.326} C_VEL
LIN {X 0,Y 402.715,Z 294.944,A -85,B 0,C 180,E1 -11231.038,E2 -11231.038} C_VEL
LIN {X 0,Y 401.8,Z 374.501,A -85,B 0,C 180,E1 -11232.472,E2 -11232.472} C_VEL
LIN {X 0,Y 401.233,Z 387.868,A -85,B 0,C 180,E1 -11232.906,E2 -11232.906} C_VEL
LIN {X 0,Y 400.604,Z 400.099,A -85,B 0,C 180,E1 -11233.502,E2 -11233.502} C_VEL
LIN {X 0,Y 399.827,Z 412.422,A -85,B 0,C 180,E1 -11234.321,E2 -11234.321} C_VEL
LIN {X 0,Y 398.984,Z 424.06,A -85,B 0,C 180,E1 -11235.332,E2 -11235.332} C_VEL
LIN {X 0,Y 398.353,Z 433.634,A -85,B 0,C 180,E1 -11236.372,E2 -11236.372} C_VEL
LIN {X 0,Y 397.762,Z 442.199,A -85,B 0,C 180,E1 -11237.5,E2 -11237.5} C_VEL
LIN {X 0,Y 397.053,Z 450.231,A -85,B 0,C 180,E1 -11238.773,E2 -11238.773} C_VEL
LIN {X 0,Y 396.53,Z 458.1,A -85,B 0,C 180,E1 -11240.307,E2 -11240.307} C_VEL
LIN {X 0,Y 396.172,Z 464.385,A -85,B 0,C 180,E1 -11241.841,E2 -11241.841} C_VEL
LIN {X 0,Y 395.933,Z 469.523,A -85,B 0,C 180,E1 -11243.426,E2 -11243.426} C_VEL
LIN {X 0,Y 395.844,Z 473.234,A -85,B 0,C 180,E1 -11244.907,E2 -11244.907} C_VEL
LIN {X 0,Y 395.775,Z 475.216,A -85,B 0,C 180,E1 -11245.927,E2 -11245.927} C_VEL
LIN {X 0,Y 395.73,Z 476.783,A -85,B 0,C 180,E1 -11246.946,E2 -11246.946} C_VEL
LIN {X 0,Y 395.763,Z 477.917,A -85,B 0,C 180,E1 -11247.965,E2 -11247.965} C_VEL
LIN {X 0,Y 395.791,Z 478.625,A -85,B 0,C 180,E1 -11248.983,E2 -11248.983} C_VEL
LIN {X 0,Y 395.791,Z 478.883,A -85,B 0,C 180,E1 -11251.017,E2 -11251.017} C_VEL
LIN {X 0,Y 395.762,Z 478.413,A -85,B 0,C 180,E1 -11252.035,E2 -11252.035} C_VEL
LIN {X 0,Y 395.774,Z 476.231,A -85,B 0,C 180,E1 -11254.073,E2 -11254.073} C_VEL
LIN {X 0,Y 395.827,Z 473.086,A -85,B 0,C 180,E1 -11255.806,E2 -11255.806} C_VEL
LIN {X 0,Y 396.094,Z 468.313,A -85,B 0,C 180,E1 -11257.647,E2 -11257.647} C_VEL
LIN {X 0,Y 396.56,Z 462.061,A -85,B 0,C 180,E1 -11259.435,E2 -11259.435} C_VEL
LIN {X 0,Y 397.146,Z 455.269,A -85,B 0,C 180,E1 -11260.967,E2 -11260.967} C_VEL
LIN {X 0,Y 398.077,Z 446.834,A -85,B 0,C 180,E1 -11262.49,E2 -11262.49} C_VEL
LIN {X 0,Y 398.897,Z 438.164,A -85,B 0,C 180,E1 -11263.76,E2 -11263.76} C_VEL
LIN {X 0,Y 399.742,Z 427.431,A -85,B 0,C 180,E1 -11265.039,E2 -11265.039} C_VEL
LIN {X 0,Y 400.721,Z 416.93,A -85,B 0,C 180,E1 -11266.035,E2 -11266.035} C_VEL
LIN {X 0,Y 401.652,Z 405.131,A -85,B 0,C 180,E1 -11266.912,E2 -11266.912} C_VEL
LIN {X 0,Y 402.458,Z 392.879,A -85,B 0,C 180,E1 -11267.597,E2 -11267.597} C_VEL
LIN {X 0,Y 403.165,Z 380.342,A -85,B 0,C 180,E1 -11268.09,E2 -11268.09} C_VEL
LIN {X 0,Y 403.561,Z 367.03,A -85,B 0,C 180,E1 -11268.408,E2 -11268.408} C_VEL
LIN {X 0,Y 404.469,Z 294.572,A -85,B 0,C 180,E1 -11269.712,E2 -11269.712} C_VEL
LIN {X 0,Y 400.126,Z 270.138,A -85,B 0,C 180,E1 -11270.423,E2 -11270.423} C_VEL
LIN {X 0,Y 399.381,Z 266.149,A -85,B 0,C 180,E1 -11270.566,E2 -11270.566} C_VEL
LIN {X 0,Y 400.851,Z 248.71,A -85,B 0,C 180,E1 -11274.258,E2 -11274.258} C_VEL
LIN {X 0,Y 398.962,Z 238.331,A -85,B 0,C 180,E1 -11276.692,E2 -11276.692} C_VEL
LIN {X 0,Y 397.131,Z 230.019,A -85,B 0,C 180,E1 -11278.76,E2 -11278.76} C_VEL
LIN {X 0,Y 397.08,Z 230.024,A -85,B 0,C 180,E1 -11282.071,E2 -11282.071} C_VEL
LIN {X 0,Y 397.12,Z 230.019,A -85,B 0,C 180,E1 -11285.503,E2 -11285.503} C_VEL
LIN {X 0,Y 397.127,Z 230.016,A -85,B 0,C 180,E1 -11288.861,E2 -11288.861} C_VEL
LIN {X 0,Y 397.065,Z 230.024,A -85,B 0,C 180,E1 -11292.268,E2 -11292.268} C_VEL
LIN {X 0,Y 397.087,Z 230.022,A -85,B 0,C 180,E1 -11295.069,E2 -11295.069} C_VEL
LIN {X 0,Y 397.062,Z 230.024,A -85,B 0,C 180,E1 -11298.022,E2 -11298.022} C_VEL
LIN {X 0,Y 397.093,Z 230.021,A -85,B 0,C 180,E1 -11301.724,E2 -11301.724} C_VEL
LIN {X 0,Y 397.125,Z 230.016,A -85,B 0,C 180,E1 -11305.507,E2 -11305.507} C_VEL
LIN {X 0,Y 397.079,Z 230.023,A -85,B 0,C 180,E1 -11309.118,E2 -11309.118} C_VEL
LIN {X 0,Y 397.138,Z 230.013,A -85,B 0,C 180,E1 -11312.606,E2 -11312.606} C_VEL
LIN {X 0,Y 397.124,Z 230.016,A -85,B 0,C 180,E1 -11315.981,E2 -11315.981} C_VEL
LIN {X 0,Y 397.14,Z 230.016,A -85,B 0,C 180,E1 -11319.705,E2 -11319.705} C_VEL
LIN {X 0,Y 397.183,Z 230.006,A -85,B 0,C 180,E1 -11322.845,E2 -11322.845} C_VEL
LIN {X 0,Y 397.23,Z 230.001,A -85,B 0,C 180,E1 -11326.703,E2 -11326.703} C_VEL
LIN {X 0,Y 397.218,Z 230.005,A -85,B 0,C 180,E1 -11329.809,E2 -11329.809} C_VEL
LIN {X 0,Y 397.354,Z 229.982,A -85,B 0,C 180,E1 -11332.888,E2 -11332.888} C_VEL
LIN {X 0,Y 397.251,Z 229.998,A -85,B 0,C 180,E1 -11334.925,E2 -11334.925} C_VEL
LIN {X 0,Y 397.446,Z 229.969,A -85,B 0,C 180,E1 -11337.973,E2 -11337.973} C_VEL
LIN {X 0,Y 397.578,Z 229.959,A -85,B 0,C 180,E1 -11340,E2 -11340} C_VEL
LIN {X 0,Y 397.369,Z 229.981,A -85,B 0,C 180,E1 -11343.042,E2 -11343.042} C_VEL
LIN {X 0,Y 397.321,Z 229.989,A -85,B 0,C 180,E1 -11346.477,E2 -11346.477} C_VEL
LIN {X 0,Y 397.236,Z 229.997,A -85,B 0,C 180,E1 -11349.162,E2 -11349.162} C_VEL
LIN {X 0,Y 397.22,Z 230,A -85,B 0,C 180,E1 -11352.258,E2 -11352.258} C_VEL
LIN {X 0,Y 397.179,Z 230.011,A -85,B 0,C 180,E1 -11355.392,E2 -11355.392} C_VEL
LIN {X 0,Y 397.158,Z 230.004,A -85,B 0,C 180,E1 -11358.574,E2 -11358.574} C_VEL
LIN {X 0,Y 397.098,Z 230.013,A -85,B 0,C 180,E1 -11361.819,E2 -11361.819} C_VEL
LIN {X 0,Y 397.156,Z 230.013,A -85,B 0,C 180,E1 -11365.132,E2 -11365.132} C_VEL
LIN {X 0,Y 397.163,Z 230.012,A -85,B 0,C 180,E1 -11367.776,E2 -11367.776} C_VEL
LIN {X 0,Y 397.08,Z 230.018,A -85,B 0,C 180,E1 -11370.883,E2 -11370.883} C_VEL
LIN {X 0,Y 397.127,Z 230.014,A -85,B 0,C 180,E1 -11374.493,E2 -11374.493} C_VEL
LIN {X 0,Y 397.101,Z 230.017,A -85,B 0,C 180,E1 -11378.276,E2 -11378.276} C_VEL
LIN {X 0,Y 397.088,Z 230.022,A -85,B 0,C 180,E1 -11380.909,E2 -11380.909} C_VEL
LIN {X 0,Y 397.102,Z 230.021,A -85,B 0,C 180,E1 -11383.649,E2 -11383.649} C_VEL
LIN {X 0,Y 397.102,Z 230.014,A -85,B 0,C 180,E1 -11386.521,E2 -11386.521} C_VEL
LIN {X 0,Y 397.088,Z 230.02,A -85,B 0,C 180,E1 -11390.42,E2 -11390.42} C_VEL
LIN {X 0,Y 397.099,Z 230.026,A -85,B 0,C 180,E1 -11393.005,E2 -11393.005} C_VEL
LIN {X 0,Y 397.121,Z 230.018,A -85,B 0,C 180,E1 -11396.282,E2 -11396.282} C_VEL
LIN {X 0,Y 397.122,Z 230.042,A -85,B 0,C 180,E1 -11399.51,E2 -11399.51} C_VEL
LIN {X 0,Y 399.358,Z 240.612,A -85,B 0,C 180,E1 -11402.21,E2 -11402.21} C_VEL
LIN {X 0,Y 399.764,Z 246.052,A -85,B 0,C 180,E1 -11403.516,E2 -11403.516} C_VEL
LIN {X 0,Y 404.633,Z 267.588,A -85,B 0,C 180,E1 -11404.219,E2 -11404.219} C_VEL
LIN {X 0,Y 404.893,Z 273.869,A -85,B 0,C 180,E1 -11404.352,E2 -11404.352} C_VEL
LIN {X 0,Y 403.56,Z 354.034,A -85,B 0,C 180,E1 -11405.808,E2 -11405.808} C_VEL
LIN {X 0,Y 403.068,Z 367.254,A -85,B 0,C 180,E1 -11406.255,E2 -11406.255} C_VEL
LIN {X 0,Y 402.449,Z 379.415,A -85,B 0,C 180,E1 -11406.864,E2 -11406.864} C_VEL
LIN {X 0,Y 401.644,Z 391.154,A -85,B 0,C 180,E1 -11407.657,E2 -11407.657} C_VEL
LIN {X 0,Y 400.73,Z 402.575,A -85,B 0,C 180,E1 -11408.659,E2 -11408.659} C_VEL
LIN {X 0,Y 399.703,Z 413.096,A -85,B 0,C 180,E1 -11409.814,E2 -11409.814} C_VEL
LIN {X 0,Y 398.971,Z 421.675,A -85,B 0,C 180,E1 -11410.981,E2 -11410.981} C_VEL
LIN {X 0,Y 398.139,Z 430.238,A -85,B 0,C 180,E1 -11412.406,E2 -11412.406} C_VEL
LIN {X 0,Y 397.309,Z 438.318,A -85,B 0,C 180,E1 -11414.087,E2 -11414.087} C_VEL
LIN {X 0,Y 396.768,Z 444.229,A -85,B 0,C 180,E1 -11415.642,E2 -11415.642} C_VEL
LIN {X 0,Y 396.363,Z 448.933,A -85,B 0,C 180,E1 -11417.219,E2 -11417.219} C_VEL
LIN {X 0,Y 396.075,Z 452.382,A -85,B 0,C 180,E1 -11418.744,E2 -11418.744} C_VEL
LIN {X 0,Y 395.847,Z 454.148,A -85,B 0,C 180,E1 -11419.773,E2 -11419.773} C_VEL
LIN {X 0,Y 395.773,Z 456.413,A -85,B 0,C 180,E1 -11421.833,E2 -11421.833} C_VEL
LIN {X 0,Y 395.772,Z 456.956,A -85,B 0,C 180,E1 -11422.859,E2 -11422.859} C_VEL
LIN {X 0,Y 395.823,Z 457.066,A -85,B 0,C 180,E1 -11423.884,E2 -11423.884} C_VEL
LIN {X 0,Y 395.751,Z 456.125,A -85,B 0,C 180,E1 -11425.927,E2 -11425.927} C_VEL
LIN {X 0,Y 395.769,Z 455.077,A -85,B 0,C 180,E1 -11426.946,E2 -11426.946} C_VEL
LIN {X 0,Y 395.887,Z 453.581,A -85,B 0,C 180,E1 -11427.965,E2 -11427.965} C_VEL
LIN {X 0,Y 395.975,Z 450.57,A -85,B 0,C 180,E1 -11429.491,E2 -11429.491} C_VEL
LIN {X 0,Y 396.17,Z 446.52,A -85,B 0,C 180,E1 -11431.016,E2 -11431.016} C_VEL
LIN {X 0,Y 396.624,Z 440.309,A -85,B 0,C 180,E1 -11432.793,E2 -11432.793} C_VEL
LIN {X 0,Y 396.654,Z 439.486,A -85,B 0,C 180,E1 -11433.002,E2 -11433.002} C_VEL
LIN {X 0,Y 396.156,Z 436.484,A -85,B 0,C 180,E1 -11433.736,E2 -11433.736} C_VEL
LIN {X 0,Y 393.73,Z 431.17,A -85,B 0,C 180,E1 -11434.901,E2 -11434.901} C_VEL
LIN {X 0,Y 391.444,Z 425.224,A -85,B 0,C 180,E1 -11436.011,E2 -11436.011} C_VEL
LIN {X 0,Y 391.165,Z 421.233,A -85,B 0,C 180,E1 -11436.648,E2 -11436.648} C_VEL
LIN {X 0,Y 392.007,Z 411.203,A -85,B 0,C 180,E1 -11437.987,E2 -11437.987} C_VEL
LIN {X 0,Y 392.839,Z 400.488,A -85,B 0,C 180,E1 -11439.136,E2 -11439.136} C_VEL
LIN {X 0,Y 393.561,Z 390.05,A -85,B 0,C 180,E1 -11440.027,E2 -11440.027} C_VEL
LIN {X 0,Y 394.199,Z 378.631,A -85,B 0,C 180,E1 -11440.789,E2 -11440.789} C_VEL
LIN {X 0,Y 394.77,Z 365.607,A -85,B 0,C 180,E1 -11441.429,E2 -11441.429} C_VEL
LIN {X 0,Y 395.084,Z 353.069,A -85,B 0,C 180,E1 -11441.842,E2 -11441.842} C_VEL
LIN {X 0,Y 396.199,Z 268.848,A -85,B 0,C 180,E1 -11443.379,E2 -11443.379} C_VEL
LIN {X 0,Y 392.044,Z 246.069,A -85,B 0,C 180,E1 -11444.02,E2 -11444.02} C_VEL
LIN {X 0,Y 392.029,Z 240.558,A -85,B 0,C 180,E1 -11445.306,E2 -11445.306} C_VEL
LIN {X 0,Y 390.143,Z 230.889,A -85,B 0,C 180,E1 -11447.757,E2 -11447.757} C_VEL
LIN {X 0,Y 390.058,Z 230.896,A -85,B 0,C 180,E1 -11451.122,E2 -11451.122} C_VEL
LIN {X 0,Y 390.064,Z 230.897,A -85,B 0,C 180,E1 -11454.482,E2 -11454.482} C_VEL
LIN {X 0,Y 390.072,Z 230.893,A -85,B 0,C 180,E1 -11458.012,E2 -11458.012} C_VEL
LIN {X 0,Y 390.026,Z 230.898,A -85,B 0,C 180,E1 -11461.504,E2 -11461.504} C_VEL
LIN {X 0,Y 390.087,Z 230.892,A -85,B 0,C 180,E1 -11465.207,E2 -11465.207} C_VEL
LIN {X 0,Y 390.07,Z 230.894,A -85,B 0,C 180,E1 -11469.218,E2 -11469.218} C_VEL
LIN {X 0,Y 390.044,Z 230.899,A -85,B 0,C 180,E1 -11472.374,E2 -11472.374} C_VEL
LIN {X 0,Y 390.045,Z 230.896,A -85,B 0,C 180,E1 -11475.354,E2 -11475.354} C_VEL
LIN {X 0,Y 390.029,Z 230.899,A -85,B 0,C 180,E1 -11478.186,E2 -11478.186} C_VEL
LIN {X 0,Y 390.088,Z 230.894,A -85,B 0,C 180,E1 -11480.907,E2 -11480.907} C_VEL
LIN {X 0,Y 390.086,Z 230.896,A -85,B 0,C 180,E1 -11484.793,E2 -11484.793} C_VEL
LIN {X 0,Y 390.025,Z 230.903,A -85,B 0,C 180,E1 -11488.496,E2 -11488.496} C_VEL
LIN {X 0,Y 390.118,Z 230.887,A -85,B 0,C 180,E1 -11492.07,E2 -11492.07} C_VEL
LIN {X 0,Y 390.077,Z 230.891,A -85,B 0,C 180,E1 -11495.519,E2 -11495.519} C_VEL
LIN {X 0,Y 390.063,Z 230.897,A -85,B 0,C 180,E1 -11498.878,E2 -11498.878} C_VEL
LIN {X 0,Y 390.127,Z 230.887,A -85,B 0,C 180,E1 -11502.166,E2 -11502.166} C_VEL
LIN {X 0,Y 390.144,Z 230.883,A -85,B 0,C 180,E1 -11505.392,E2 -11505.392} C_VEL
LIN {X 0,Y 390.148,Z 230.889,A -85,B 0,C 180,E1 -11508.571,E2 -11508.571} C_VEL
LIN {X 0,Y 390.259,Z 230.87,A -85,B 0,C 180,E1 -11512.084,E2 -11512.084} C_VEL
LIN {X 0,Y 390.218,Z 230.878,A -85,B 0,C 180,E1 -11514.833,E2 -11514.833} C_VEL
LIN {X 0,Y 390.419,Z 230.849,A -85,B 0,C 180,E1 -11517.937,E2 -11517.937} C_VEL
LIN {X 0,Y 390.547,Z 230.834,A -85,B 0,C 180,E1 -11520,E2 -11520} C_VEL
LIN {X 0,Y 390.303,Z 230.865,A -85,B 0,C 180,E1 -11523.097,E2 -11523.097} C_VEL
LIN {X 0,Y 390.33,Z 230.862,A -85,B 0,C 180,E1 -11526.202,E2 -11526.202} C_VEL
LIN {X 0,Y 390.315,Z 230.865,A -85,B 0,C 180,E1 -11528.282,E2 -11528.282} C_VEL
LIN {X 0,Y 390.171,Z 230.885,A -85,B 0,C 180,E1 -11532.483,E2 -11532.483} C_VEL
LIN {X 0,Y 390.14,Z 230.883,A -85,B 0,C 180,E1 -11535.677,E2 -11535.677} C_VEL
LIN {X 0,Y 390.103,Z 230.891,A -85,B 0,C 180,E1 -11538.922,E2 -11538.922} C_VEL
LIN {X 0,Y 390.038,Z 230.899,A -85,B 0,C 180,E1 -11542.234,E2 -11542.234} C_VEL
LIN {X 0,Y 390.084,Z 230.891,A -85,B 0,C 180,E1 -11545.733,E2 -11545.733} C_VEL
LIN {X 0,Y 390.034,Z 230.898,A -85,B 0,C 180,E1 -11549.112,E2 -11549.112} C_VEL
LIN {X 0,Y 390.043,Z 230.901,A -85,B 0,C 180,E1 -11552.722,E2 -11552.722} C_VEL
LIN {X 0,Y 390.055,Z 230.894,A -85,B 0,C 180,E1 -11555.825,E2 -11555.825} C_VEL
LIN {X 0,Y 390.038,Z 230.897,A -85,B 0,C 180,E1 -11559.213,E2 -11559.213} C_VEL
LIN {X 0,Y 390.039,Z 230.901,A -85,B 0,C 180,E1 -11562.374,E2 -11562.374} C_VEL
LIN {X 0,Y 390.044,Z 230.896,A -85,B 0,C 180,E1 -11565.354,E2 -11565.354} C_VEL
LIN {X 0,Y 390.025,Z 230.901,A -85,B 0,C 180,E1 -11568.186,E2 -11568.186} C_VEL
LIN {X 0,Y 390.088,Z 230.893,A -85,B 0,C 180,E1 -11570.907,E2 -11570.907} C_VEL
LIN {X 0,Y 390.086,Z 230.894,A -85,B 0,C 180,E1 -11574.793,E2 -11574.793} C_VEL
LIN {X 0,Y 390.025,Z 230.905,A -85,B 0,C 180,E1 -11578.496,E2 -11578.496} C_VEL
LIN {X 0,Y 390.133,Z 230.903,A -85,B 0,C 180,E1 -11582.217,E2 -11582.217} C_VEL
LIN {X 0,Y 392.517,Z 243.363,A -85,B 0,C 180,E1 -11585.117,E2 -11585.117} C_VEL
LIN {X 0,Y 393.007,Z 247.066,A -85,B 0,C 180,E1 -11585.95,E2 -11585.95} C_VEL
LIN {X 0,Y 391.928,Z 262.677,A -85,B 0,C 180,E1 -11589.258,E2 -11589.258} C_VEL
LIN {X 0,Y 391.631,Z 266.195,A -85,B 0,C 180,E1 -11589.996,E2 -11589.996} C_VEL
LIN {X 0,Y 395.907,Z 295.221,A -85,B 0,C 180,E1 -11590.747,E2 -11590.747} C_VEL
LIN {X 0,Y 394.933,Z 375.28,A -85,B 0,C 180,E1 -11592.224,E2 -11592.224} C_VEL
LIN {X 0,Y 394.309,Z 389.088,A -85,B 0,C 180,E1 -11592.697,E2 -11592.697} C_VEL
LIN {X 0,Y 393.606,Z 401.476,A -85,B 0,C 180,E1 -11593.333,E2 -11593.333} C_VEL
LIN {X 0,Y 392.834,Z 413.36,A -85,B 0,C 180,E1 -11594.167,E2 -11594.167} C_VEL
LIN {X 0,Y 391.97,Z 424.79,A -85,B 0,C 180,E1 -11595.197,E2 -11595.197} C_VEL
LIN {X 0,Y 391.29,Z 434.888,A -85,B 0,C 180,E1 -11596.338,E2 -11596.338} C_VEL
LIN {X 0,Y 390.639,Z 443.518,A -85,B 0,C 180,E1 -11597.532,E2 -11597.532} C_VEL
LIN {X 0,Y 389.837,Z 452.642,A -85,B 0,C 180,E1 -11599.088,E2 -11599.088} C_VEL
LIN {X 0,Y 389.353,Z 459.997,A -85,B 0,C 180,E1 -11600.651,E2 -11600.651} C_VEL
LIN {X 0,Y 389.017,Z 465.886,A -85,B 0,C 180,E1 -11602.213,E2 -11602.213} C_VEL
LIN {X 0,Y 388.795,Z 470.658,A -85,B 0,C 180,E1 -11603.828,E2 -11603.828} C_VEL
LIN {X 0,Y 388.743,Z 472.963,A -85,B 0,C 180,E1 -11604.814,E2 -11604.814} C_VEL
LIN {X 0,Y 388.7,Z 474.958,A -85,B 0,C 180,E1 -11605.853,E2 -11605.853} C_VEL
LIN {X 0,Y 388.637,Z 476.536,A -85,B 0,C 180,E1 -11606.89,E2 -11606.89} C_VEL
LIN {X 0,Y 388.662,Z 477.692,A -85,B 0,C 180,E1 -11607.927,E2 -11607.927} C_VEL
LIN {X 0,Y 388.703,Z 478.412,A -85,B 0,C 180,E1 -11608.964,E2 -11608.964} C_VEL
LIN {X 0,Y 388.708,Z 478.745,A -85,B 0,C 180,E1 -11610,E2 -11610} C_VEL
LIN {X 0,Y 388.703,Z 478.692,A -85,B 0,C 180,E1 -11611.036,E2 -11611.036} C_VEL
LIN {X 0,Y 388.66,Z 478.242,A -85,B 0,C 180,E1 -11612.073,E2 -11612.073} C_VEL
LIN {X 0,Y 388.699,Z 476.085,A -85,B 0,C 180,E1 -11614.147,E2 -11614.147} C_VEL
LIN {X 0,Y 388.74,Z 474.407,A -85,B 0,C 180,E1 -11615.186,E2 -11615.186} C_VEL
LIN {X 0,Y 388.852,Z 471.041,A -85,B 0,C 180,E1 -11616.747,E2 -11616.747} C_VEL
LIN {X 0,Y 389.193,Z 466.612,A -85,B 0,C 180,E1 -11618.306,E2 -11618.306} C_VEL
LIN {X 0,Y 389.724,Z 459.927,A -85,B 0,C 180,E1 -11620.127,E2 -11620.127} C_VEL
LIN {X 0,Y 390.435,Z 452.641,A -85,B 0,C 180,E1 -11621.684,E2 -11621.684} C_VEL
LIN {X 0,Y 391.444,Z 443.617,A -85,B 0,C 180,E1 -11623.233,E2 -11623.233} C_VEL
LIN {X 0,Y 392.336,Z 434.302,A -85,B 0,C 180,E1 -11624.524,E2 -11624.524} C_VEL
LIN {X 0,Y 393.143,Z 425.252,A -85,B 0,C 180,E1 -11625.554,E2 -11625.554} C_VEL
LIN {X 0,Y 394.182,Z 414.08,A -85,B 0,C 180,E1 -11626.575,E2 -11626.575} C_VEL
LIN {X 0,Y 395.063,Z 403.528,A -85,B 0,C 180,E1 -11627.336,E2 -11627.336} C_VEL
LIN {X 0,Y 395.927,Z 390.844,A -85,B 0,C 180,E1 -11628.031,E2 -11628.031} C_VEL
LIN {X 0,Y 396.558,Z 378.265,A -85,B 0,C 180,E1 -11628.502,E2 -11628.502} C_VEL
LIN {X 0,Y 397.024,Z 361.129,A -85,B 0,C 180,E1 -11628.87,E2 -11628.87} C_VEL
LIN {X 0,Y 397.793,Z 294.94,A -85,B 0,C 180,E1 -11630.086,E2 -11630.086} C_VEL
LIN {X 0,Y 393.415,Z 270.43,A -85,B 0,C 180,E1 -11630.819,E2 -11630.819} C_VEL
LIN {X 0,Y 392.531,Z 265.95,A -85,B 0,C 180,E1 -11630.983,E2 -11630.983} C_VEL
LIN {X 0,Y 393.867,Z 250.884,A -85,B 0,C 180,E1 -11634.23,E2 -11634.23} C_VEL
LIN {X 0,Y 393.471,Z 246.994,A -85,B 0,C 180,E1 -11635.128,E2 -11635.128} C_VEL
LIN {X 0,Y 391.215,Z 235.823,A -85,B 0,C 180,E1 -11637.845,E2 -11637.845} C_VEL
LIN {X 0,Y 390.081,Z 230.893,A -85,B 0,C 180,E1 -11639.108,E2 -11639.108} C_VEL
LIN {X 0,Y 390.044,Z 230.9,A -85,B 0,C 180,E1 -11642.721,E2 -11642.721} C_VEL
LIN {X 0,Y 390.057,Z 230.899,A -85,B 0,C 180,E1 -11645.825,E2 -11645.825} C_VEL
LIN {X 0,Y 390.068,Z 230.899,A -85,B 0,C 180,E1 -11649.218,E2 -11649.218} C_VEL
LIN {X 0,Y 390.04,Z 230.899,A -85,B 0,C 180,E1 -11652.373,E2 -11652.373} C_VEL
LIN {X 0,Y 390.044,Z 230.902,A -85,B 0,C 180,E1 -11655.354,E2 -11655.354} C_VEL
LIN {X 0,Y 390.024,Z 230.9,A -85,B 0,C 180,E1 -11658.186,E2 -11658.186} C_VEL
LIN {X 0,Y 390.059,Z 230.896,A -85,B 0,C 180,E1 -11660.904,E2 -11660.904} C_VEL
LIN {X 0,Y 390.085,Z 230.892,A -85,B 0,C 180,E1 -11664.793,E2 -11664.793} C_VEL
LIN {X 0,Y 390.024,Z 230.899,A -85,B 0,C 180,E1 -11668.496,E2 -11668.496} C_VEL
LIN {X 0,Y 390.075,Z 230.894,A -85,B 0,C 180,E1 -11672.067,E2 -11672.067} C_VEL
LIN {X 0,Y 390.062,Z 230.896,A -85,B 0,C 180,E1 -11675.518,E2 -11675.518} C_VEL
LIN {X 0,Y 390.056,Z 230.892,A -85,B 0,C 180,E1 -11678.878,E2 -11678.878} C_VEL
LIN {X 0,Y 390.112,Z 230.886,A -85,B 0,C 180,E1 -11682.166,E2 -11682.166} C_VEL
LIN {X 0,Y 390.145,Z 230.888,A -85,B 0,C 180,E1 -11685.393,E2 -11685.393} C_VEL
LIN {X 0,Y 390.148,Z 230.877,A -85,B 0,C 180,E1 -11688.571,E2 -11688.571} C_VEL
LIN {X 0,Y 390.309,Z 230.859,A -85,B 0,C 180,E1 -11692.031,E2 -11692.031} C_VEL
LIN {X 0,Y 390.223,Z 230.873,A -85,B 0,C 180,E1 -11694.834,E2 -11694.834} C_VEL
LIN {X 0,Y 390.414,Z 230.845,A -85,B 0,C 180,E1 -11697.937,E2 -11697.937} C_VEL
LIN {X 0,Y 390.547,Z 230.834,A -85,B 0,C 180,E1 -11700,E2 -11700} C_VEL
LIN {X 0,Y 390.303,Z 230.861,A -85,B 0,C 180,E1 -11703.097,E2 -11703.097} C_VEL
LIN {X 0,Y 390.28,Z 230.866,A -85,B 0,C 180,E1 -11706.468,E2 -11706.468} C_VEL
LIN {X 0,Y 390.194,Z 230.876,A -85,B 0,C 180,E1 -11709.329,E2 -11709.329} C_VEL
LIN {X 0,Y 390.172,Z 230.877,A -85,B 0,C 180,E1 -11712.483,E2 -11712.483} C_VEL
LIN {X 0,Y 390.14,Z 230.887,A -85,B 0,C 180,E1 -11715.677,E2 -11715.677} C_VEL
LIN {X 0,Y 390.103,Z 230.884,A -85,B 0,C 180,E1 -11718.922,E2 -11718.922} C_VEL
LIN {X 0,Y 390.04,Z 230.89,A -85,B 0,C 180,E1 -11722.234,E2 -11722.234} C_VEL
LIN {X 0,Y 390.119,Z 230.884,A -85,B 0,C 180,E1 -11725.743,E2 -11725.743} C_VEL
LIN {X 0,Y 390.06,Z 230.898,A -85,B 0,C 180,E1 -11729.11,E2 -11729.11} C_VEL
LIN {X 0,Y 390.044,Z 230.897,A -85,B 0,C 180,E1 -11732.722,E2 -11732.722} C_VEL
LIN {X 0,Y 390.057,Z 230.894,A -85,B 0,C 180,E1 -11735.825,E2 -11735.825} C_VEL
LIN {X 0,Y 390.068,Z 230.896,A -85,B 0,C 180,E1 -11739.218,E2 -11739.218} C_VEL
LIN {X 0,Y 390.04,Z 230.898,A -85,B 0,C 180,E1 -11742.374,E2 -11742.374} C_VEL
LIN {X 0,Y 390.046,Z 230.901,A -85,B 0,C 180,E1 -11745.355,E2 -11745.355} C_VEL
LIN {X 0,Y 390.025,Z 230.904,A -85,B 0,C 180,E1 -11748.186,E2 -11748.186} C_VEL
LIN {X 0,Y 390.061,Z 230.898,A -85,B 0,C 180,E1 -11750.904,E2 -11750.904} C_VEL
LIN {X 0,Y 390.087,Z 230.897,A -85,B 0,C 180,E1 -11754.793,E2 -11754.793} C_VEL
LIN {X 0,Y 390.028,Z 230.9,A -85,B 0,C 180,E1 -11758.496,E2 -11758.496} C_VEL
LIN {X 0,Y 390.07,Z 230.992,A -85,B 0,C 180,E1 -11759.179,E2 -11759.179} C_VEL
LIN {X 0,Y 392.29,Z 241.299,A -85,B 0,C 180,E1 -11761.869,E2 -11761.869} C_VEL
LIN {X 0,Y 392.893,Z 246.225,A -85,B 0,C 180,E1 -11763.091,E2 -11763.091} C_VEL
LIN {X 0,Y 397.565,Z 266.211,A -85,B 0,C 180,E1 -11763.778,E2 -11763.778} C_VEL
LIN {X 0,Y 398.337,Z 270.551,A -85,B 0,C 180,E1 -11763.908,E2 -11763.908} C_VEL
LIN {X 0,Y 396.94,Z 354.022,A -85,B 0,C 180,E1 -11765.448,E2 -11765.448} C_VEL
LIN {X 0,Y 396.425,Z 367.311,A -85,B 0,C 180,E1 -11765.901,E2 -11765.901} C_VEL
LIN {X 0,Y 395.771,Z 379.507,A -85,B 0,C 180,E1 -11766.519,E2 -11766.519} C_VEL
LIN {X 0,Y 394.983,Z 390.454,A -85,B 0,C 180,E1 -11767.26,E2 -11767.26} C_VEL
LIN {X 0,Y 394.016,Z 402.134,A -85,B 0,C 180,E1 -11768.286,E2 -11768.286} C_VEL
LIN {X 0,Y 392.936,Z 412.698,A -85,B 0,C 180,E1 -11769.451,E2 -11769.451} C_VEL
LIN {X 0,Y 392.162,Z 421.377,A -85,B 0,C 180,E1 -11770.638,E2 -11770.638} C_VEL
LIN {X 0,Y 391.316,Z 429.339,A -85,B 0,C 180,E1 -11771.952,E2 -11771.952} C_VEL
LIN {X 0,Y 390.49,Z 437.079,A -85,B 0,C 180,E1 -11773.533,E2 -11773.533} C_VEL
LIN {X 0,Y 389.95,Z 442.354,A -85,B 0,C 180,E1 -11774.851,E2 -11774.851} C_VEL
LIN {X 0,Y 389.487,Z 447.437,A -85,B 0,C 180,E1 -11776.433,E2 -11776.433} C_VEL
LIN {X 0,Y 389.103,Z 451.364,A -85,B 0,C 180,E1 -11778.012,E2 -11778.012} C_VEL
LIN {X 0,Y 388.795,Z 454.245,A -85,B 0,C 180,E1 -11779.586,E2 -11779.586} C_VEL
LIN {X 0,Y 388.677,Z 456.554,A -85,B 0,C 180,E1 -11781.683,E2 -11781.683} C_VEL
LIN {X 0,Y 388.67,Z 457.123,A -85,B 0,C 180,E1 -11782.728,E2 -11782.728} C_VEL
LIN {X 0,Y 388.731,Z 457.251,A -85,B 0,C 180,E1 -11783.917,E2 -11783.917} C_VEL
LIN {X 0,Y 388.674,Z 456.376,A -85,B 0,C 180,E1 -11785.852,E2 -11785.852} C_VEL
LIN {X 0,Y 388.671,Z 455.353,A -85,B 0,C 180,E1 -11786.89,E2 -11786.89} C_VEL
LIN {X 0,Y 388.782,Z 453.902,A -85,B 0,C 180,E1 -11787.928,E2 -11787.928} C_VEL
LIN {X 0,Y 388.886,Z 450.938,A -85,B 0,C 180,E1 -11789.482,E2 -11789.482} C_VEL
LIN {X 0,Y 389.084,Z 446.937,A -85,B 0,C 180,E1 -11791.035,E2 -11791.035} C_VEL
LIN {X 0,Y 389.563,Z 440.782,A -85,B 0,C 180,E1 -11792.844,E2 -11792.844} C_VEL
LIN {X 0,Y 390.026,Z 434.096,A -85,B 0,C 180,E1 -11794.392,E2 -11794.392} C_VEL
LIN {X 0,Y 390.813,Z 425.787,A -85,B 0,C 180,E1 -11795.935,E2 -11795.935} C_VEL
LIN {X 0,Y 391.165,Z 421.233,A -85,B 0,C 180,E1 -11796.648,E2 -11796.648} C_VEL
LIN {X 0,Y 390.747,Z 418.5,A -85,B 0,C 180,E1 -11797.067,E2 -11797.067} C_VEL
LIN {X 0,Y 388.309,Z 414.171,A -85,B 0,C 180,E1 -11797.742,E2 -11797.742} C_VEL
LIN {X 0,Y 385.882,Z 409.646,A -85,B 0,C 180,E1 -11798.394,E2 -11798.394} C_VEL
LIN {X 0,Y 385.474,Z 406.549,A -85,B 0,C 180,E1 -11798.764,E2 -11798.764} C_VEL
LIN {X 0,Y 386.311,Z 395.82,A -85,B 0,C 180,E1 -11799.82,E2 -11799.82} C_VEL
LIN {X 0,Y 387.035,Z 384.032,A -85,B 0,C 180,E1 -11800.727,E2 -11800.727} C_VEL
LIN {X 0,Y 387.709,Z 371.766,A -85,B 0,C 180,E1 -11801.435,E2 -11801.435} C_VEL
LIN {X 0,Y 388.124,Z 358.428,A -85,B 0,C 180,E1 -11801.979,E2 -11801.979} C_VEL
LIN {X 0,Y 388.458,Z 343.678,A -85,B 0,C 180,E1 -11802.318,E2 -11802.318} C_VEL
LIN {X 0,Y 389.419,Z 269.693,A -85,B 0,C 180,E1 -11803.677,E2 -11803.677} C_VEL
LIN {X 0,Y 385.122,Z 246.264,A -85,B 0,C 180,E1 -11804.35,E2 -11804.35} C_VEL
LIN {X 0,Y 385.104,Z 242.081,A -85,B 0,C 180,E1 -11805.344,E2 -11805.344} C_VEL
LIN {X 0,Y 383.084,Z 231.769,A -85,B 0,C 180,E1 -11807.981,E2 -11807.981} C_VEL
LIN {X 0,Y 382.995,Z 231.774,A -85,B 0,C 180,E1 -11811.531,E2 -11811.531} C_VEL
LIN {X 0,Y 383.031,Z 231.773,A -85,B 0,C 180,E1 -11814.962,E2 -11814.962} C_VEL
LIN {X 0,Y 383.005,Z 231.777,A -85,B 0,C 180,E1 -11818.496,E2 -11818.496} C_VEL
LIN {X 0,Y 383.011,Z 231.773,A -85,B 0,C 180,E1 -11822.149,E2 -11822.149} C_VEL
LIN {X 0,Y 383.02,Z 231.777,A -85,B 0,C 180,E1 -11824.668,E2 -11824.668} C_VEL
LIN {X 0,Y 383.001,Z 231.773,A -85,B 0,C 180,E1 -11827.903,E2 -11827.903} C_VEL
LIN {X 0,Y 382.985,Z 231.775,A -85,B 0,C 180,E1 -11831.347,E2 -11831.347} C_VEL
LIN {X 0,Y 382.997,Z 231.776,A -85,B 0,C 180,E1 -11834.303,E2 -11834.303} C_VEL
LIN {X 0,Y 383.011,Z 231.773,A -85,B 0,C 180,E1 -11837.24,E2 -11837.24} C_VEL
LIN {X 0,Y 383.01,Z 231.776,A -85,B 0,C 180,E1 -11840.414,E2 -11840.414} C_VEL
LIN {X 0,Y 383.026,Z 231.771,A -85,B 0,C 180,E1 -11844.044,E2 -11844.044} C_VEL
LIN {X 0,Y 382.988,Z 231.774,A -85,B 0,C 180,E1 -11847.578,E2 -11847.578} C_VEL
LIN {X 0,Y 382.993,Z 231.777,A -85,B 0,C 180,E1 -11850.3,E2 -11850.3} C_VEL
LIN {X 0,Y 383.08,Z 231.764,A -85,B 0,C 180,E1 -11854.021,E2 -11854.021} C_VEL
LIN {X 0,Y 383.013,Z 231.772,A -85,B 0,C 180,E1 -11857.335,E2 -11857.335} C_VEL
LIN {X 0,Y 383.059,Z 231.772,A -85,B 0,C 180,E1 -11860.716,E2 -11860.716} C_VEL
LIN {X 0,Y 383.081,Z 231.764,A -85,B 0,C 180,E1 -11864.026,E2 -11864.026} C_VEL
LIN {X 0,Y 383.137,Z 231.757,A -85,B 0,C 180,E1 -11867.284,E2 -11867.284} C_VEL
LIN {X 0,Y 383.144,Z 231.761,A -85,B 0,C 180,E1 -11870.498,E2 -11870.498} C_VEL
LIN {X 0,Y 383.256,Z 231.741,A -85,B 0,C 180,E1 -11873.683,E2 -11873.683} C_VEL
LIN {X 0,Y 383.386,Z 231.725,A -85,B 0,C 180,E1 -11877.899,E2 -11877.899} C_VEL
LIN {X 0,Y 383.516,Z 231.71,A -85,B 0,C 180,E1 -11880,E2 -11880} C_VEL
LIN {X 0,Y 383.239,Z 231.745,A -85,B 0,C 180,E1 -11883.154,E2 -11883.154} C_VEL
LIN {X 0,Y 383.288,Z 231.741,A -85,B 0,C 180,E1 -11886.316,E2 -11886.316} C_VEL
LIN {X 0,Y 383.261,Z 231.745,A -85,B 0,C 180,E1 -11888.436,E2 -11888.436} C_VEL
LIN {X 0,Y 383.097,Z 231.761,A -85,B 0,C 180,E1 -11891.642,E2 -11891.642} C_VEL
LIN {X 0,Y 383.111,Z 231.763,A -85,B 0,C 180,E1 -11894.882,E2 -11894.882} C_VEL
LIN {X 0,Y 383.053,Z 231.769,A -85,B 0,C 180,E1 -11898.174,E2 -11898.174} C_VEL
LIN {X 0,Y 382.993,Z 231.774,A -85,B 0,C 180,E1 -11901.531,E2 -11901.531} C_VEL
LIN {X 0,Y 383.029,Z 231.772,A -85,B 0,C 180,E1 -11904.962,E2 -11904.962} C_VEL
LIN {X 0,Y 382.986,Z 231.781,A -85,B 0,C 180,E1 -11908.497,E2 -11908.497} C_VEL
LIN {X 0,Y 383.009,Z 231.774,A -85,B 0,C 180,E1 -11912.15,E2 -11912.15} C_VEL
LIN {X 0,Y 383.018,Z 231.776,A -85,B 0,C 180,E1 -11914.668,E2 -11914.668} C_VEL
LIN {X 0,Y 382.994,Z 231.774,A -85,B 0,C 180,E1 -11917.903,E2 -11917.903} C_VEL
LIN {X 0,Y 382.965,Z 231.778,A -85,B 0,C 180,E1 -11921.35,E2 -11921.35} C_VEL
LIN {X 0,Y 382.995,Z 231.778,A -85,B 0,C 180,E1 -11924.303,E2 -11924.303} C_VEL
LIN {X 0,Y 383.011,Z 231.772,A -85,B 0,C 180,E1 -11927.24,E2 -11927.24} C_VEL
LIN {X 0,Y 383.009,Z 231.777,A -85,B 0,C 180,E1 -11930.415,E2 -11930.415} C_VEL
LIN {X 0,Y 383.025,Z 231.772,A -85,B 0,C 180,E1 -11934.045,E2 -11934.045} C_VEL
LIN {X 0,Y 382.988,Z 231.774,A -85,B 0,C 180,E1 -11937.578,E2 -11937.578} C_VEL
LIN {X 0,Y 382.993,Z 231.778,A -85,B 0,C 180,E1 -11940.3,E2 -11940.3} C_VEL
LIN {X 0,Y 383.085,Z 231.835,A -85,B 0,C 180,E1 -11941.973,E2 -11941.973} C_VEL
LIN {X 0,Y 385.25,Z 242.933,A -85,B 0,C 180,E1 -11944.615,E2 -11944.615} C_VEL
LIN {X 0,Y 385.947,Z 247.068,A -85,B 0,C 180,E1 -11945.573,E2 -11945.573} C_VEL
LIN {X 0,Y 385.462,Z 255.867,A -85,B 0,C 180,E1 -11947.487,E2 -11947.487} C_VEL
LIN {X 0,Y 384.738,Z 266.044,A -85,B 0,C 180,E1 -11949.674,E2 -11949.674} C_VEL
LIN {X 0,Y 389.128,Z 296.162,A -85,B 0,C 180,E1 -11950.46,E2 -11950.46} C_VEL
LIN {X 0,Y 388.106,Z 374.879,A -85,B 0,C 180,E1 -11951.934,E2 -11951.934} C_VEL
LIN {X 0,Y 387.494,Z 388.76,A -85,B 0,C 180,E1 -11952.417,E2 -11952.417} C_VEL
LIN {X 0,Y 386.819,Z 400.657,A -85,B 0,C 180,E1 -11953.032,E2 -11953.032} C_VEL
LIN {X 0,Y 385.996,Z 412.699,A -85,B 0,C 180,E1 -11953.879,E2 -11953.879} C_VEL
LIN {X 0,Y 385.081,Z 424.214,A -85,B 0,C 180,E1 -11954.926,E2 -11954.926} C_VEL
LIN {X 0,Y 384.363,Z 433.991,A -85,B 0,C 180,E1 -11956.038,E2 -11956.038} C_VEL
LIN {X 0,Y 383.658,Z 443.075,A -85,B 0,C 180,E1 -11957.302,E2 -11957.302} C_VEL
LIN {X 0,Y 382.826,Z 452.248,A -85,B 0,C 180,E1 -11958.886,E2 -11958.886} C_VEL
LIN {X 0,Y 382.313,Z 459.639,A -85,B 0,C 180,E1 -11960.477,E2 -11960.477} C_VEL
LIN {X 0,Y 381.94,Z 465.558,A -85,B 0,C 180,E1 -11962.068,E2 -11962.068} C_VEL
LIN {X 0,Y 381.699,Z 470.736,A -85,B 0,C 180,E1 -11963.865,E2 -11963.865} C_VEL
LIN {X 0,Y 381.625,Z 474.698,A -85,B 0,C 180,E1 -11965.776,E2 -11965.776} C_VEL
LIN {X 0,Y 381.548,Z 476.287,A -85,B 0,C 180,E1 -11966.832,E2 -11966.832} C_VEL
LIN {X 0,Y 381.561,Z 477.464,A -85,B 0,C 180,E1 -11967.889,E2 -11967.889} C_VEL
LIN {X 0,Y 381.617,Z 478.199,A -85,B 0,C 180,E1 -11968.945,E2 -11968.945} C_VEL
LIN {X 0,Y 381.639,Z 478.544,A -85,B 0,C 180,E1 -11970,E2 -11970} C_VEL
LIN {X 0,Y 381.602,Z 478.501,A -85,B 0,C 180,E1 -11971.055,E2 -11971.055} C_VEL
LIN {X 0,Y 381.558,Z 478.069,A -85,B 0,C 180,E1 -11972.111,E2 -11972.111} C_VEL
LIN {X 0,Y 381.624,Z 475.94,A -85,B 0,C 180,E1 -11974.225,E2 -11974.225} C_VEL
LIN {X 0,Y 381.678,Z 472.674,A -85,B 0,C 180,E1 -11976.105,E2 -11976.105} C_VEL
LIN {X 0,Y 381.997,Z 468.145,A -85,B 0,C 180,E1 -11977.931,E2 -11977.931} C_VEL
LIN {X 0,Y 382.524,Z 461.955,A -85,B 0,C 180,E1 -11979.785,E2 -11979.785} C_VEL
LIN {X 0,Y 383.14,Z 455.229,A -85,B 0,C 180,E1 -11981.373,E2 -11981.373} C_VEL
LIN {X 0,Y 384.197,Z 446.898,A -85,B 0,C 180,E1 -11982.949,E2 -11982.949} C_VEL
LIN {X 0,Y 385.141,Z 437.457,A -85,B 0,C 180,E1 -11984.383,E2 -11984.383} C_VEL
LIN {X 0,Y 386.015,Z 428.034,A -85,B 0,C 180,E1 -11985.551,E2 -11985.551} C_VEL
LIN {X 0,Y 387.094,Z 417.368,A -85,B 0,C 180,E1 -11986.616,E2 -11986.616} C_VEL
LIN {X 0,Y 388.139,Z 405.893,A -85,B 0,C 180,E1 -11987.519,E2 -11987.519} C_VEL
LIN {X 0,Y 389.019,Z 394.009,A -85,B 0,C 180,E1 -11988.226,E2 -11988.226} C_VEL
LIN {X 0,Y 389.867,Z 380.273,A -85,B 0,C 180,E1 -11988.798,E2 -11988.798} C_VEL
LIN {X 0,Y 390.286,Z 367.499,A -85,B 0,C 180,E1 -11989.122,E2 -11989.122} C_VEL
LIN {X 0,Y 391.275,Z 296.244,A -85,B 0,C 180,E1 -11990.447,E2 -11990.447} C_VEL
LIN {X 0,Y 386.882,Z 271.664,A -85,B 0,C 180,E1 -11991.202,E2 -11991.202} C_VEL
LIN {X 0,Y 385.754,Z 265.724,A -85,B 0,C 180,E1 -11991.419,E2 -11991.419} C_VEL
LIN {X 0,Y 386.979,Z 252.137,A -85,B 0,C 180,E1 -11994.404,E2 -11994.404} C_VEL
LIN {X 0,Y 386.328,Z 247.119,A -85,B 0,C 180,E1 -11995.598,E2 -11995.598} C_VEL
LIN {X 0,Y 383.905,Z 235.458,A -85,B 0,C 180,E1 -11998.512,E2 -11998.512} C_VEL
LIN {X 0,Y 383.031,Z 231.768,A -85,B 0,C 180,E1 -11999.47,E2 -11999.47} C_VEL
LIN {X 0,Y 383.004,Z 231.776,A -85,B 0,C 180,E1 -12003.401,E2 -12003.401} C_VEL
LIN {X 0,Y 383.033,Z 231.772,A -85,B 0,C 180,E1 -12006.164,E2 -12006.164} C_VEL
LIN {X 0,Y 383.008,Z 231.776,A -85,B 0,C 180,E1 -12009.958,E2 -12009.958} C_VEL
LIN {X 0,Y 383.006,Z 231.776,A -85,B 0,C 180,E1 -12012.779,E2 -12012.779} C_VEL
LIN {X 0,Y 382.997,Z 231.778,A -85,B 0,C 180,E1 -12015.789,E2 -12015.789} C_VEL
LIN {X 0,Y 382.966,Z 231.78,A -85,B 0,C 180,E1 -12018.8,E2 -12018.8} C_VEL
LIN {X 0,Y 382.994,Z 231.774,A -85,B 0,C 180,E1 -12022.097,E2 -12022.097} C_VEL
LIN {X 0,Y 383.018,Z 231.776,A -85,B 0,C 180,E1 -12025.332,E2 -12025.332} C_VEL
LIN {X 0,Y 382.983,Z 231.779,A -85,B 0,C 180,E1 -12029.081,E2 -12029.081} C_VEL
LIN {X 0,Y 383.019,Z 231.772,A -85,B 0,C 180,E1 -12032.695,E2 -12032.695} C_VEL
LIN {X 0,Y 383.018,Z 231.772,A -85,B 0,C 180,E1 -12036.192,E2 -12036.192} C_VEL
LIN {X 0,Y 383.056,Z 231.768,A -85,B 0,C 180,E1 -12039.599,E2 -12039.599} C_VEL
LIN {X 0,Y 383.095,Z 231.761,A -85,B 0,C 180,E1 -12042.931,E2 -12042.931} C_VEL
LIN {X 0,Y 383.126,Z 231.757,A -85,B 0,C 180,E1 -12046.464,E2 -12046.464} C_VEL
LIN {X 0,Y 383.152,Z 231.754,A -85,B 0,C 180,E1 -12050.498,E2 -12050.498} C_VEL
LIN {X 0,Y 383.284,Z 231.738,A -85,B 0,C 180,E1 -12053.684,E2 -12053.684} C_VEL
LIN {X 0,Y 383.38,Z 231.721,A -85,B 0,C 180,E1 -12057.899,E2 -12057.899} C_VEL
LIN {X 0,Y 383.516,Z 231.71,A -85,B 0,C 180,E1 -12060,E2 -12060} C_VEL
LIN {X 0,Y 383.24,Z 231.741,A -85,B 0,C 180,E1 -12063.154,E2 -12063.154} C_VEL
LIN {X 0,Y 383.244,Z 231.742,A -85,B 0,C 180,E1 -12066.455,E2 -12066.455} C_VEL
LIN {X 0,Y 383.144,Z 231.757,A -85,B 0,C 180,E1 -12069.502,E2 -12069.502} C_VEL
LIN {X 0,Y 383.127,Z 231.755,A -85,B 0,C 180,E1 -12073.536,E2 -12073.536} C_VEL
LIN {X 0,Y 383.095,Z 231.764,A -85,B 0,C 180,E1 -12077.069,E2 -12077.069} C_VEL
LIN {X 0,Y 383.03,Z 231.769,A -85,B 0,C 180,E1 -12080.647,E2 -12080.647} C_VEL
LIN {X 0,Y 383.033,Z 231.771,A -85,B 0,C 180,E1 -12083.808,E2 -12083.808} C_VEL
LIN {X 0,Y 383.08,Z 231.758,A -85,B 0,C 180,E1 -12086.124,E2 -12086.124} C_VEL
LIN {X 0,Y 382.993,Z 231.774,A -85,B 0,C 180,E1 -12089.7,E2 -12089.7} C_VEL
LIN {X 0,Y 383.005,Z 231.775,A -85,B 0,C 180,E1 -12093.401,E2 -12093.401} C_VEL
LIN {X 0,Y 383.033,Z 231.767,A -85,B 0,C 180,E1 -12096.165,E2 -12096.165} C_VEL
LIN {X 0,Y 383.009,Z 231.775,A -85,B 0,C 180,E1 -12099.959,E2 -12099.959} C_VEL
LIN {X 0,Y 383.007,Z 231.775,A -85,B 0,C 180,E1 -12102.779,E2 -12102.779} C_VEL
LIN {X 0,Y 382.998,Z 231.774,A -85,B 0,C 180,E1 -12105.789,E2 -12105.789} C_VEL
LIN {X 0,Y 382.967,Z 231.785,A -85,B 0,C 180,E1 -12108.8,E2 -12108.8} C_VEL
LIN {X 0,Y 382.996,Z 231.781,A -85,B 0,C 180,E1 -12112.098,E2 -12112.098} C_VEL
LIN {X 0,Y 383.02,Z 231.778,A -85,B 0,C 180,E1 -12115.332,E2 -12115.332} C_VEL
LIN {X 0,Y 383.025,Z 231.881,A -85,B 0,C 180,E1 -12118.817,E2 -12118.817} C_VEL
LIN {X 0,Y 384.978,Z 240.778,A -85,B 0,C 180,E1 -12121.196,E2 -12121.196} C_VEL
LIN {X 0,Y 386.012,Z 246.684,A -85,B 0,C 180,E1 -12122.674,E2 -12122.674} C_VEL
LIN {X 0,Y 390.553,Z 264.926,A -85,B 0,C 180,E1 -12123.325,E2 -12123.325} C_VEL
LIN {X 0,Y 391.803,Z 272.115,A -85,B 0,C 180,E1 -12123.543,E2 -12123.543} C_VEL
LIN {X 0,Y 390.332,Z 354.038,A -85,B 0,C 180,E1 -12125.075,E2 -12125.075} C_VEL
LIN {X 0,Y 389.776,Z 367.381,A -85,B 0,C 180,E1 -12125.534,E2 -12125.534} C_VEL
LIN {X 0,Y 389.117,Z 379.612,A -85,B 0,C 180,E1 -12126.164,E2 -12126.164} C_VEL
LIN {X 0,Y 388.237,Z 391.083,A -85,B 0,C 180,E1 -12126.954,E2 -12126.954} C_VEL
LIN {X 0,Y 387.198,Z 403.01,A -85,B 0,C 180,E1 -12128.032,E2 -12128.032} C_VEL
LIN {X 0,Y 386.077,Z 413.387,A -85,B 0,C 180,E1 -12129.208,E2 -12129.208} C_VEL
LIN {X 0,Y 385.155,Z 422.836,A -85,B 0,C 180,E1 -12130.548,E2 -12130.548} C_VEL
LIN {X 0,Y 384.235,Z 431.203,A -85,B 0,C 180,E1 -12132.014,E2 -12132.014} C_VEL
LIN {X 0,Y 383.321,Z 439.217,A -85,B 0,C 180,E1 -12133.764,E2 -12133.764} C_VEL
LIN {X 0,Y 382.805,Z 444.122,A -85,B 0,C 180,E1 -12135.106,E2 -12135.106} C_VEL
LIN {X 0,Y 382.257,Z 449.642,A -85,B 0,C 180,E1 -12137.018,E2 -12137.018} C_VEL
LIN {X 0,Y 381.963,Z 452.481,A -85,B 0,C 180,E1 -12138.323,E2 -12138.323} C_VEL
LIN {X 0,Y 381.751,Z 454.336,A -85,B 0,C 180,E1 -12139.391,E2 -12139.391} C_VEL
LIN {X 0,Y 381.599,Z 456.696,A -85,B 0,C 180,E1 -12141.527,E2 -12141.527} C_VEL
LIN {X 0,Y 381.583,Z 457.287,A -85,B 0,C 180,E1 -12142.592,E2 -12142.592} C_VEL
LIN {X 0,Y 381.658,Z 457.44,A -85,B 0,C 180,E1 -12143.924,E2 -12143.924} C_VEL
LIN {X 0,Y 381.598,Z 456.627,A -85,B 0,C 180,E1 -12145.775,E2 -12145.775} C_VEL
LIN {X 0,Y 381.577,Z 455.627,A -85,B 0,C 180,E1 -12146.832,E2 -12146.832} C_VEL
LIN {X 0,Y 381.678,Z 454.219,A -85,B 0,C 180,E1 -12147.889,E2 -12147.889} C_VEL
LIN {X 0,Y 381.8,Z 451.294,A -85,B 0,C 180,E1 -12149.473,E2 -12149.473} C_VEL
LIN {X 0,Y 382.002,Z 447.341,A -85,B 0,C 180,E1 -12151.054,E2 -12151.054} C_VEL
LIN {X 0,Y 382.414,Z 442.249,A -85,B 0,C 180,E1 -12152.633,E2 -12152.633} C_VEL
LIN {X 0,Y 382.9,Z 435.847,A -85,B 0,C 180,E1 -12154.21,E2 -12154.21} C_VEL
LIN {X 0,Y 383.6,Z 427.879,A -85,B 0,C 180,E1 -12155.783,E2 -12155.783} C_VEL
LIN {X 0,Y 384.367,Z 419.752,A -85,B 0,C 180,E1 -12157.09,E2 -12157.09} C_VEL
LIN {X 0,Y 385.21,Z 409.852,A -85,B 0,C 180,E1 -12158.393,E2 -12158.393} C_VEL
LIN {X 0,Y 385.474,Z 406.549,A -85,B 0,C 180,E1 -12158.764,E2 -12158.764} C_VEL
LIN {X 0,Y 385.204,Z 401.815,A -85,B 0,C 180,E1 -12159.293,E2 -12159.293} C_VEL
LIN {X 0,Y 382.955,Z 393.949,A -85,B 0,C 180,E1 -12160.139,E2 -12160.139} C_VEL
LIN {X 0,Y 380.709,Z 385.674,A -85,B 0,C 180,E1 -12160.887,E2 -12160.887} C_VEL
LIN {X 0,Y 380.431,Z 380.307,A -85,B 0,C 180,E1 -12161.253,E2 -12161.253} C_VEL
LIN {X 0,Y 381.056,Z 367.042,A -85,B 0,C 180,E1 -12161.946,E2 -12161.946} C_VEL
LIN {X 0,Y 381.427,Z 354.241,A -85,B 0,C 180,E1 -12162.396,E2 -12162.396} C_VEL
LIN {X 0,Y 382.637,Z 270.358,A -85,B 0,C 180,E1 -12163.988,E2 -12163.988} C_VEL
LIN {X 0,Y 378.211,Z 246.497,A -85,B 0,C 180,E1 -12164.683,E2 -12164.683} C_VEL
LIN {X 0,Y 378.003,Z 242.587,A -85,B 0,C 180,E1 -12165.64,E2 -12165.64} C_VEL
LIN {X 0,Y 376.062,Z 232.644,A -85,B 0,C 180,E1 -12168.229,E2 -12168.229} C_VEL
LIN {X 0,Y 375.96,Z 232.65,A -85,B 0,C 180,E1 -12171.954,E2 -12171.954} C_VEL
LIN {X 0,Y 375.978,Z 232.648,A -85,B 0,C 180,E1 -12175.463,E2 -12175.463} C_VEL
LIN {X 0,Y 375.931,Z 232.656,A -85,B 0,C 180,E1 -12179.082,E2 -12179.082} C_VEL
LIN {X 0,Y 375.96,Z 232.65,A -85,B 0,C 180,E1 -12181.562,E2 -12181.562} C_VEL
LIN {X 0,Y 375.959,Z 232.65,A -85,B 0,C 180,E1 -12185.415,E2 -12185.415} C_VEL
LIN {X 0,Y 375.975,Z 232.65,A -85,B 0,C 180,E1 -12188.27,E2 -12188.27} C_VEL
LIN {X 0,Y 375.936,Z 232.653,A -85,B 0,C 180,E1 -12191.6,E2 -12191.6} C_VEL
LIN {X 0,Y 375.928,Z 232.655,A -85,B 0,C 180,E1 -12195.268,E2 -12195.268} C_VEL
LIN {X 0,Y 375.932,Z 232.657,A -85,B 0,C 180,E1 -12198.4,E2 -12198.4} C_VEL
LIN {X 0,Y 375.973,Z 232.648,A -85,B 0,C 180,E1 -12201.73,E2 -12201.73} C_VEL
LIN {X 0,Y 375.981,Z 232.648,A -85,B 0,C 180,E1 -12205.332,E2 -12205.332} C_VEL
LIN {X 0,Y 375.959,Z 232.654,A -85,B 0,C 180,E1 -12208.438,E2 -12208.438} C_VEL
LIN {X 0,Y 375.984,Z 232.649,A -85,B 0,C 180,E1 -12212.14,E2 -12212.14} C_VEL
LIN {X 0,Y 376.006,Z 232.65,A -85,B 0,C 180,E1 -12214.539,E2 -12214.539} C_VEL
LIN {X 0,Y 375.968,Z 232.65,A -85,B 0,C 180,E1 -12218.046,E2 -12218.046} C_VEL
LIN {X 0,Y 376.008,Z 232.644,A -85,B 0,C 180,E1 -12221.473,E2 -12221.473} C_VEL
LIN {X 0,Y 376.059,Z 232.642,A -85,B 0,C 180,E1 -12224.832,E2 -12224.832} C_VEL
LIN {X 0,Y 376.05,Z 232.641,A -85,B 0,C 180,E1 -12228.136,E2 -12228.136} C_VEL
LIN {X 0,Y 376.174,Z 232.624,A -85,B 0,C 180,E1 -12231.968,E2 -12231.968} C_VEL
LIN {X 0,Y 376.16,Z 232.632,A -85,B 0,C 180,E1 -12234.64,E2 -12234.64} C_VEL
LIN {X 0,Y 376.352,Z 232.601,A -85,B 0,C 180,E1 -12237.86,E2 -12237.86} C_VEL
LIN {X 0,Y 376.486,Z 232.585,A -85,B 0,C 180,E1 -12240,E2 -12240} C_VEL
LIN {X 0,Y 376.349,Z 232.603,A -85,B 0,C 180,E1 -12242.14,E2 -12242.14} C_VEL
LIN {X 0,Y 376.247,Z 232.619,A -85,B 0,C 180,E1 -12246.435,E2 -12246.435} C_VEL
LIN {X 0,Y 376.206,Z 232.626,A -85,B 0,C 180,E1 -12248.595,E2 -12248.595} C_VEL
LIN {X 0,Y 376.049,Z 232.639,A -85,B 0,C 180,E1 -12251.863,E2 -12251.863} C_VEL
LIN {X 0,Y 376.059,Z 232.639,A -85,B 0,C 180,E1 -12255.167,E2 -12255.167} C_VEL
LIN {X 0,Y 376.003,Z 232.651,A -85,B 0,C 180,E1 -12258.527,E2 -12258.527} C_VEL
LIN {X 0,Y 375.957,Z 232.651,A -85,B 0,C 180,E1 -12261.955,E2 -12261.955} C_VEL
LIN {X 0,Y 375.966,Z 232.649,A -85,B 0,C 180,E1 -12265.464,E2 -12265.464} C_VEL
LIN {X 0,Y 375.92,Z 232.657,A -85,B 0,C 180,E1 -12269.083,E2 -12269.083} C_VEL
LIN {X 0,Y 375.957,Z 232.65,A -85,B 0,C 180,E1 -12271.562,E2 -12271.562} C_VEL
LIN {X 0,Y 375.957,Z 232.65,A -85,B 0,C 180,E1 -12275.416,E2 -12275.416} C_VEL
LIN {X 0,Y 375.937,Z 232.656,A -85,B 0,C 180,E1 -12278.263,E2 -12278.263} C_VEL
LIN {X 0,Y 375.92,Z 232.655,A -85,B 0,C 180,E1 -12281.598,E2 -12281.598} C_VEL
LIN {X 0,Y 375.927,Z 232.659,A -85,B 0,C 180,E1 -12284.731,E2 -12284.731} C_VEL
LIN {X 0,Y 375.925,Z 232.659,A -85,B 0,C 180,E1 -12288.401,E2 -12288.401} C_VEL
LIN {X 0,Y 375.963,Z 232.651,A -85,B 0,C 180,E1 -12291.911,E2 -12291.911} C_VEL
LIN {X 0,Y 375.981,Z 232.648,A -85,B 0,C 180,E1 -12295.333,E2 -12295.333} C_VEL
LIN {X 0,Y 375.959,Z 232.656,A -85,B 0,C 180,E1 -12298.438,E2 -12298.438} C_VEL
LIN {X 0,Y 375.988,Z 232.687,A -85,B 0,C 180,E1 -12301.697,E2 -12301.697} C_VEL
LIN {X 0,Y 377.941,Z 242.496,A -85,B 0,C 180,E1 -12304.088,E2 -12304.088} C_VEL
LIN {X 0,Y 379.013,Z 248.479,A -85,B 0,C 180,E1 -12305.508,E2 -12305.508} C_VEL
LIN {X 0,Y 378.299,Z 259.315,A -85,B 0,C 180,E1 -12307.901,E2 -12307.901} C_VEL
LIN {X 0,Y 377.816,Z 265.858,A -85,B 0,C 180,E1 -12309.333,E2 -12309.333} C_VEL
LIN {X 0,Y 382.37,Z 296.91,A -85,B 0,C 180,E1 -12310.16,E2 -12310.16} C_VEL
LIN {X 0,Y 381.314,Z 374.458,A -85,B 0,C 180,E1 -12311.636,E2 -12311.636} C_VEL
LIN {X 0,Y 380.728,Z 387.649,A -85,B 0,C 180,E1 -12312.094,E2 -12312.094} C_VEL
LIN {X 0,Y 380.034,Z 399.788,A -85,B 0,C 180,E1 -12312.72,E2 -12312.72} C_VEL
LIN {X 0,Y 379.148,Z 412.028,A -85,B 0,C 180,E1 -12313.58,E2 -12313.58} C_VEL
LIN {X 0,Y 378.185,Z 423.63,A -85,B 0,C 180,E1 -12314.644,E2 -12314.644} C_VEL
LIN {X 0,Y 377.394,Z 433.925,A -85,B 0,C 180,E1 -12315.832,E2 -12315.832} C_VEL
LIN {X 0,Y 376.682,Z 442.621,A -85,B 0,C 180,E1 -12317.062,E2 -12317.062} C_VEL
LIN {X 0,Y 375.799,Z 451.85,A -85,B 0,C 180,E1 -12318.676,E2 -12318.676} C_VEL
LIN {X 0,Y 375.255,Z 459.275,A -85,B 0,C 180,E1 -12320.296,E2 -12320.296} C_VEL
LIN {X 0,Y 374.878,Z 465.228,A -85,B 0,C 180,E1 -12321.917,E2 -12321.917} C_VEL
LIN {X 0,Y 374.632,Z 469.917,A -85,B 0,C 180,E1 -12323.537,E2 -12323.537} C_VEL
LIN {X 0,Y 374.545,Z 473.487,A -85,B 0,C 180,E1 -12325.156,E2 -12325.156} C_VEL
LIN {X 0,Y 374.463,Z 476.038,A -85,B 0,C 180,E1 -12326.772,E2 -12326.772} C_VEL
LIN {X 0,Y 374.461,Z 477.233,A -85,B 0,C 180,E1 -12327.849,E2 -12327.849} C_VEL
LIN {X 0,Y 374.517,Z 477.985,A -85,B 0,C 180,E1 -12328.925,E2 -12328.925} C_VEL
LIN {X 0,Y 374.554,Z 478.341,A -85,B 0,C 180,E1 -12330,E2 -12330} C_VEL
LIN {X 0,Y 374.503,Z 478.31,A -85,B 0,C 180,E1 -12331.075,E2 -12331.075} C_VEL
LIN {X 0,Y 374.457,Z 477.893,A -85,B 0,C 180,E1 -12332.151,E2 -12332.151} C_VEL
LIN {X 0,Y 374.46,Z 477.047,A -85,B 0,C 180,E1 -12333.228,E2 -12333.228} C_VEL
LIN {X 0,Y 374.529,Z 475.796,A -85,B 0,C 180,E1 -12334.305,E2 -12334.305} C_VEL
LIN {X 0,Y 374.586,Z 472.852,A -85,B 0,C 180,E1 -12336.072,E2 -12336.072} C_VEL
LIN {X 0,Y 374.934,Z 468.058,A -85,B 0,C 180,E1 -12338.082,E2 -12338.082} C_VEL
LIN {X 0,Y 375.513,Z 461.907,A -85,B 0,C 180,E1 -12339.969,E2 -12339.969} C_VEL
LIN {X 0,Y 376.167,Z 455.214,A -85,B 0,C 180,E1 -12341.586,E2 -12341.586} C_VEL
LIN {X 0,Y 377.255,Z 446.928,A -85,B 0,C 180,E1 -12343.192,E2 -12343.192} C_VEL
LIN {X 0,Y 378.248,Z 437.432,A -85,B 0,C 180,E1 -12344.668,E2 -12344.668} C_VEL
LIN {X 0,Y 379.326,Z 426.901,A -85,B 0,C 180,E1 -12345.984,E2 -12345.984} C_VEL
LIN {X 0,Y 380.483,Z 416.173,A -85,B 0,C 180,E1 -12347.052,E2 -12347.052} C_VEL
LIN {X 0,Y 381.582,Z 404.317,A -85,B 0,C 180,E1 -12347.969,E2 -12347.969} C_VEL
LIN {X 0,Y 382.514,Z 392.001,A -85,B 0,C 180,E1 -12348.686,E2 -12348.686} C_VEL
LIN {X 0,Y 383.267,Z 379.355,A -85,B 0,C 180,E1 -12349.203,E2 -12349.203} C_VEL
LIN {X 0,Y 383.697,Z 366.135,A -85,B 0,C 180,E1 -12349.529,E2 -12349.529} C_VEL
LIN {X 0,Y 384.697,Z 296.774,A -85,B 0,C 180,E1 -12350.841,E2 -12350.841} C_VEL
LIN {X 0,Y 380.048,Z 271.296,A -85,B 0,C 180,E1 -12351.652,E2 -12351.652} C_VEL
LIN {X 0,Y 378.942,Z 265.57,A -85,B 0,C 180,E1 -12351.857,E2 -12351.857} C_VEL
LIN {X 0,Y 380.072,Z 253.651,A -85,B 0,C 180,E1 -12354.526,E2 -12354.526} C_VEL
LIN {X 0,Y 379.606,Z 249.63,A -85,B 0,C 180,E1 -12355.496,E2 -12355.496} C_VEL
LIN {X 0,Y 377.371,Z 238.571,A -85,B 0,C 180,E1 -12358.299,E2 -12358.299} C_VEL
LIN {X 0,Y 375.955,Z 232.65,A -85,B 0,C 180,E1 -12359.927,E2 -12359.927} C_VEL
LIN {X 0,Y 375.95,Z 232.655,A -85,B 0,C 180,E1 -12362.828,E2 -12362.828} C_VEL
LIN {X 0,Y 375.958,Z 232.654,A -85,B 0,C 180,E1 -12365.415,E2 -12365.415} C_VEL
LIN {X 0,Y 375.973,Z 232.651,A -85,B 0,C 180,E1 -12368.27,E2 -12368.27} C_VEL
LIN {X 0,Y 375.934,Z 232.659,A -85,B 0,C 180,E1 -12371.6,E2 -12371.6} C_VEL
LIN {X 0,Y 375.927,Z 232.66,A -85,B 0,C 180,E1 -12375.269,E2 -12375.269} C_VEL
LIN {X 0,Y 375.921,Z 232.657,A -85,B 0,C 180,E1 -12378.402,E2 -12378.402} C_VEL
LIN {X 0,Y 375.954,Z 232.652,A -85,B 0,C 180,E1 -12381.91,E2 -12381.91} C_VEL
LIN {X 0,Y 375.98,Z 232.652,A -85,B 0,C 180,E1 -12385.333,E2 -12385.333} C_VEL
LIN {X 0,Y 375.958,Z 232.651,A -85,B 0,C 180,E1 -12388.438,E2 -12388.438} C_VEL
LIN {X 0,Y 375.958,Z 232.652,A -85,B 0,C 180,E1 -12392.138,E2 -12392.138} C_VEL
LIN {X 0,Y 375.977,Z 232.643,A -85,B 0,C 180,E1 -12394.537,E2 -12394.537} C_VEL
LIN {X 0,Y 375.958,Z 232.648,A -85,B 0,C 180,E1 -12398.045,E2 -12398.045} C_VEL
LIN {X 0,Y 376.003,Z 232.65,A -85,B 0,C 180,E1 -12401.473,E2 -12401.473} C_VEL
LIN {X 0,Y 376.06,Z 232.637,A -85,B 0,C 180,E1 -12404.833,E2 -12404.833} C_VEL
LIN {X 0,Y 376.05,Z 232.634,A -85,B 0,C 180,E1 -12408.137,E2 -12408.137} C_VEL
LIN {X 0,Y 376.221,Z 232.615,A -85,B 0,C 180,E1 -12411.918,E2 -12411.918} C_VEL
LIN {X 0,Y 376.169,Z 232.623,A -85,B 0,C 180,E1 -12414.64,E2 -12414.64} C_VEL
LIN {X 0,Y 376.345,Z 232.597,A -85,B 0,C 180,E1 -12417.86,E2 -12417.86} C_VEL
LIN {X 0,Y 376.486,Z 232.586,A -85,B 0,C 180,E1 -12420,E2 -12420} C_VEL
LIN {X 0,Y 376.35,Z 232.598,A -85,B 0,C 180,E1 -12422.141,E2 -12422.141} C_VEL
LIN {X 0,Y 376.214,Z 232.619,A -85,B 0,C 180,E1 -12426.438,E2 -12426.438} C_VEL
LIN {X 0,Y 376.114,Z 232.635,A -85,B 0,C 180,E1 -12429.682,E2 -12429.682} C_VEL
LIN {X 0,Y 376.091,Z 232.632,A -85,B 0,C 180,E1 -12433.658,E2 -12433.658} C_VEL
LIN {X 0,Y 376.033,Z 232.64,A -85,B 0,C 180,E1 -12437.4,E2 -12437.4} C_VEL
LIN {X 0,Y 375.979,Z 232.648,A -85,B 0,C 180,E1 -12440.832,E2 -12440.832} C_VEL
LIN {X 0,Y 375.994,Z 232.646,A -85,B 0,C 180,E1 -12444.282,E2 -12444.282} C_VEL
LIN {X 0,Y 376.021,Z 232.638,A -85,B 0,C 180,E1 -12446.652,E2 -12446.652} C_VEL
LIN {X 0,Y 375.966,Z 232.647,A -85,B 0,C 180,E1 -12450.313,E2 -12450.313} C_VEL
LIN {X 0,Y 375.961,Z 232.652,A -85,B 0,C 180,E1 -12454.112,E2 -12454.112} C_VEL
LIN {X 0,Y 375.954,Z 232.65,A -85,B 0,C 180,E1 -12456.741,E2 -12456.741} C_VEL
LIN {X 0,Y 375.989,Z 232.65,A -85,B 0,C 180,E1 -12459.971,E2 -12459.971} C_VEL
LIN {X 0,Y 375.931,Z 232.658,A -85,B 0,C 180,E1 -12463.766,E2 -12463.766} C_VEL
LIN {X 0,Y 375.935,Z 232.651,A -85,B 0,C 180,E1 -12466.811,E2 -12466.811} C_VEL
LIN {X 0,Y 375.938,Z 232.655,A -85,B 0,C 180,E1 -12470.534,E2 -12470.534} C_VEL
LIN {X 0,Y 375.965,Z 232.659,A -85,B 0,C 180,E1 -12473.496,E2 -12473.496} C_VEL
LIN {X 0,Y 375.962,Z 232.656,A -85,B 0,C 180,E1 -12475.889,E2 -12475.889} C_VEL
LIN {X 0,Y 375.979,Z 232.775,A -85,B 0,C 180,E1 -12478.44,E2 -12478.44} C_VEL
LIN {X 0,Y 378.372,Z 243.752,A -85,B 0,C 180,E1 -12481.427,E2 -12481.427} C_VEL
LIN {X 0,Y 378.925,Z 246.725,A -85,B 0,C 180,E1 -12482.202,E2 -12482.202} C_VEL
LIN {X 0,Y 381.325,Z 254.595,A -85,B 0,C 180,E1 -12482.523,E2 -12482.523} C_VEL
LIN {X 0,Y 385.208,Z 271.973,A -85,B 0,C 180,E1 -12483.125,E2 -12483.125} C_VEL
LIN {X 0,Y 383.744,Z 354.075,A -85,B 0,C 180,E1 -12484.689,E2 -12484.689} C_VEL
LIN {X 0,Y 383.166,Z 367.469,A -85,B 0,C 180,E1 -12485.156,E2 -12485.156} C_VEL
LIN {X 0,Y 382.471,Z 379.726,A -85,B 0,C 180,E1 -12485.795,E2 -12485.795} C_VEL
LIN {X 0,Y 381.489,Z 392.023,A -85,B 0,C 180,E1 -12486.666,E2 -12486.666} C_VEL
LIN {X 0,Y 380.45,Z 403.324,A -85,B 0,C 180,E1 -12487.712,E2 -12487.712} C_VEL
LIN {X 0,Y 379.218,Z 414.079,A -85,B 0,C 180,E1 -12488.957,E2 -12488.957} C_VEL
LIN {X 0,Y 378.367,Z 422.582,A -85,B 0,C 180,E1 -12490.185,E2 -12490.185} C_VEL
LIN {X 0,Y 377.43,Z 430.385,A -85,B 0,C 180,E1 -12491.545,E2 -12491.545} C_VEL
LIN {X 0,Y 376.524,Z 437.986,A -85,B 0,C 180,E1 -12493.183,E2 -12493.183} C_VEL
LIN {X 0,Y 375.843,Z 444.072,A -85,B 0,C 180,E1 -12494.824,E2 -12494.824} C_VEL
LIN {X 0,Y 375.315,Z 448.872,A -85,B 0,C 180,E1 -12496.464,E2 -12496.464} C_VEL
LIN {X 0,Y 374.915,Z 452.533,A -85,B 0,C 180,E1 -12498.1,E2 -12498.1} C_VEL
LIN {X 0,Y 374.713,Z 454.419,A -85,B 0,C 180,E1 -12499.19,E2 -12499.19} C_VEL
LIN {X 0,Y 374.551,Z 455.839,A -85,B 0,C 180,E1 -12500.278,E2 -12500.278} C_VEL
LIN {X 0,Y 374.495,Z 457.451,A -85,B 0,C 180,E1 -12502.451,E2 -12502.451} C_VEL
LIN {X 0,Y 374.566,Z 457.625,A -85,B 0,C 180,E1 -12503.96,E2 -12503.96} C_VEL
LIN {X 0,Y 374.523,Z 456.878,A -85,B 0,C 180,E1 -12505.695,E2 -12505.695} C_VEL
LIN {X 0,Y 374.574,Z 454.526,A -85,B 0,C 180,E1 -12507.849,E2 -12507.849} C_VEL
LIN {X 0,Y 374.717,Z 451.638,A -85,B 0,C 180,E1 -12509.463,E2 -12509.463} C_VEL
LIN {X 0,Y 374.922,Z 447.733,A -85,B 0,C 180,E1 -12511.074,E2 -12511.074} C_VEL
LIN {X 0,Y 375.359,Z 442.699,A -85,B 0,C 180,E1 -12512.683,E2 -12512.683} C_VEL
LIN {X 0,Y 375.84,Z 436.376,A -85,B 0,C 180,E1 -12514.29,E2 -12514.29} C_VEL
LIN {X 0,Y 376.562,Z 428.476,A -85,B 0,C 180,E1 -12515.892,E2 -12515.892} C_VEL
LIN {X 0,Y 377.54,Z 418.656,A -85,B 0,C 180,E1 -12517.487,E2 -12517.487} C_VEL
LIN {X 0,Y 378.421,Z 408.371,A -85,B 0,C 180,E1 -12518.813,E2 -12518.813} C_VEL
LIN {X 0,Y 379.363,Z 396.782,A -85,B 0,C 180,E1 -12520.002,E2 -12520.002} C_VEL
LIN {X 0,Y 380.132,Z 385.286,A -85,B 0,C 180,E1 -12520.924,E2 -12520.924} C_VEL
LIN {X 0,Y 380.431,Z 380.307,A -85,B 0,C 180,E1 -12521.253,E2 -12521.253} C_VEL
LIN {X 0,Y 380.199,Z 374.831,A -85,B 0,C 180,E1 -12521.593,E2 -12521.593} C_VEL
LIN {X 0,Y 377.759,Z 365.914,A -85,B 0,C 180,E1 -12522.143,E2 -12522.143} C_VEL
LIN {X 0,Y 375.23,Z 356.816,A -85,B 0,C 180,E1 -12522.6,E2 -12522.6} C_VEL
LIN {X 0,Y 374.739,Z 351.061,A -85,B 0,C 180,E1 -12522.778,E2 -12522.778} C_VEL
LIN {X 0,Y 375.942,Z 271.578,A -85,B 0,C 180,E1 -12524.295,E2 -12524.295} C_VEL
LIN {X 0,Y 371.314,Z 246.654,A -85,B 0,C 180,E1 -12525.046,E2 -12525.046} C_VEL
LIN {X 0,Y 370.637,Z 241.976,A -85,B 0,C 180,E1 -12526.242,E2 -12526.242} C_VEL
LIN {X 0,Y 369.002,Z 233.523,A -85,B 0,C 180,E1 -12528.468,E2 -12528.468} C_VEL
LIN {X 0,Y 368.925,Z 233.53,A -85,B 0,C 180,E1 -12532.396,E2 -12532.396} C_VEL
LIN {X 0,Y 368.961,Z 233.522,A -85,B 0,C 180,E1 -12535.983,E2 -12535.983} C_VEL
LIN {X 0,Y 368.902,Z 233.529,A -85,B 0,C 180,E1 -12539.691,E2 -12539.691} C_VEL
LIN {X 0,Y 368.899,Z 233.532,A -85,B 0,C 180,E1 -12543.043,E2 -12543.043} C_VEL
LIN {X 0,Y 368.919,Z 233.529,A -85,B 0,C 180,E1 -12546.197,E2 -12546.197} C_VEL
LIN {X 0,Y 368.904,Z 233.532,A -85,B 0,C 180,E1 -12548.953,E2 -12548.953} C_VEL
LIN {X 0,Y 368.882,Z 233.532,A -85,B 0,C 180,E1 -12552.009,E2 -12552.009} C_VEL
LIN {X 0,Y 368.885,Z 233.533,A -85,B 0,C 180,E1 -12555.176,E2 -12555.176} C_VEL
LIN {X 0,Y 368.881,Z 233.534,A -85,B 0,C 180,E1 -12558.177,E2 -12558.177} C_VEL
LIN {X 0,Y 368.906,Z 233.529,A -85,B 0,C 180,E1 -12561.36,E2 -12561.36} C_VEL
LIN {X 0,Y 368.937,Z 233.526,A -85,B 0,C 180,E1 -12565.146,E2 -12565.146} C_VEL
LIN {X 0,Y 368.93,Z 233.528,A -85,B 0,C 180,E1 -12569.046,E2 -12569.046} C_VEL
LIN {X 0,Y 368.963,Z 233.526,A -85,B 0,C 180,E1 -12572.796,E2 -12572.796} C_VEL
LIN {X 0,Y 368.945,Z 233.525,A -85,B 0,C 180,E1 -12576.113,E2 -12576.113} C_VEL
LIN {X 0,Y 368.936,Z 233.525,A -85,B 0,C 180,E1 -12579.947,E2 -12579.947} C_VEL
LIN {X 0,Y 368.976,Z 233.52,A -85,B 0,C 180,E1 -12583.399,E2 -12583.399} C_VEL
LIN {X 0,Y 369.059,Z 233.514,A -85,B 0,C 180,E1 -12586.79,E2 -12586.79} C_VEL
LIN {X 0,Y 369.064,Z 233.511,A -85,B 0,C 180,E1 -12590.131,E2 -12590.131} C_VEL
LIN {X 0,Y 369.174,Z 233.495,A -85,B 0,C 180,E1 -12593.441,E2 -12593.441} C_VEL
LIN {X 0,Y 369.317,Z 233.478,A -85,B 0,C 180,E1 -12597.819,E2 -12597.819} C_VEL
LIN {X 0,Y 369.455,Z 233.461,A -85,B 0,C 180,E1 -12600,E2 -12600} C_VEL
LIN {X 0,Y 369.314,Z 233.48,A -85,B 0,C 180,E1 -12602.181,E2 -12602.181} C_VEL
LIN {X 0,Y 369.209,Z 233.497,A -85,B 0,C 180,E1 -12606.558,E2 -12606.558} C_VEL
LIN {X 0,Y 369.138,Z 233.505,A -85,B 0,C 180,E1 -12608.761,E2 -12608.761} C_VEL
LIN {X 0,Y 369.005,Z 233.518,A -85,B 0,C 180,E1 -12612.093,E2 -12612.093} C_VEL
LIN {X 0,Y 368.998,Z 233.517,A -85,B 0,C 180,E1 -12615.465,E2 -12615.465} C_VEL
LIN {X 0,Y 368.954,Z 233.526,A -85,B 0,C 180,E1 -12618.894,E2 -12618.894} C_VEL
LIN {X 0,Y 368.922,Z 233.531,A -85,B 0,C 180,E1 -12622.396,E2 -12622.396} C_VEL
LIN {X 0,Y 368.943,Z 233.525,A -85,B 0,C 180,E1 -12625.984,E2 -12625.984} C_VEL
LIN {X 0,Y 368.896,Z 233.53,A -85,B 0,C 180,E1 -12629.692,E2 -12629.692} C_VEL
LIN {X 0,Y 368.897,Z 233.532,A -85,B 0,C 180,E1 -12633.043,E2 -12633.043} C_VEL
LIN {X 0,Y 368.916,Z 233.53,A -85,B 0,C 180,E1 -12636.197,E2 -12636.197} C_VEL
LIN {X 0,Y 368.875,Z 233.535,A -85,B 0,C 180,E1 -12638.957,E2 -12638.957} C_VEL
LIN {X 0,Y 368.872,Z 233.534,A -85,B 0,C 180,E1 -12642.008,E2 -12642.008} C_VEL
LIN {X 0,Y 368.88,Z 233.533,A -85,B 0,C 180,E1 -12645.176,E2 -12645.176} C_VEL
LIN {X 0,Y 368.875,Z 233.535,A -85,B 0,C 180,E1 -12648.177,E2 -12648.177} C_VEL
LIN {X 0,Y 368.905,Z 233.529,A -85,B 0,C 180,E1 -12651.361,E2 -12651.361} C_VEL
LIN {X 0,Y 368.937,Z 233.526,A -85,B 0,C 180,E1 -12655.147,E2 -12655.147} C_VEL
LIN {X 0,Y 368.93,Z 233.532,A -85,B 0,C 180,E1 -12659.047,E2 -12659.047} C_VEL
LIN {X 0,Y 368.972,Z 233.613,A -85,B 0,C 180,E1 -12661.434,E2 -12661.434} C_VEL
LIN {X 0,Y 370.943,Z 243.438,A -85,B 0,C 180,E1 -12663.881,E2 -12663.881} C_VEL
LIN {X 0,Y 372.08,Z 249.911,A -85,B 0,C 180,E1 -12665.446,E2 -12665.446} C_VEL
LIN {X 0,Y 371.333,Z 260.195,A -85,B 0,C 180,E1 -12667.757,E2 -12667.757} C_VEL
LIN {X 0,Y 370.92,Z 265.663,A -85,B 0,C 180,E1 -12668.977,E2 -12668.977} C_VEL
LIN {X 0,Y 375.595,Z 297.426,A -85,B 0,C 180,E1 -12669.845,E2 -12669.845} C_VEL
LIN {X 0,Y 374.507,Z 374.012,A -85,B 0,C 180,E1 -12671.325,E2 -12671.325} C_VEL
LIN {X 0,Y 373.918,Z 387.289,A -85,B 0,C 180,E1 -12671.792,E2 -12671.792} C_VEL
LIN {X 0,Y 373.138,Z 400.036,A -85,B 0,C 180,E1 -12672.461,E2 -12672.461} C_VEL
LIN {X 0,Y 372.308,Z 411.349,A -85,B 0,C 180,E1 -12673.269,E2 -12673.269} C_VEL
LIN {X 0,Y 371.28,Z 423.039,A -85,B 0,C 180,E1 -12674.351,E2 -12674.351} C_VEL
LIN {X 0,Y 370.48,Z 433.092,A -85,B 0,C 180,E1 -12675.522,E2 -12675.522} C_VEL
LIN {X 0,Y 369.703,Z 442.153,A -85,B 0,C 180,E1 -12676.814,E2 -12676.814} C_VEL
LIN {X 0,Y 368.963,Z 450.066,A -85,B 0,C 180,E1 -12678.184,E2 -12678.184} C_VEL
LIN {X 0,Y 368.308,Z 457.784,A -85,B 0,C 180,E1 -12679.834,E2 -12679.834} C_VEL
LIN {X 0,Y 367.836,Z 464.896,A -85,B 0,C 180,E1 -12681.761,E2 -12681.761} C_VEL
LIN {X 0,Y 367.564,Z 469.615,A -85,B 0,C 180,E1 -12683.412,E2 -12683.412} C_VEL
LIN {X 0,Y 367.446,Z 473.211,A -85,B 0,C 180,E1 -12685.062,E2 -12685.062} C_VEL
LIN {X 0,Y 367.381,Z 475.788,A -85,B 0,C 180,E1 -12686.71,E2 -12686.71} C_VEL
LIN {X 0,Y 367.362,Z 476.999,A -85,B 0,C 180,E1 -12687.807,E2 -12687.807} C_VEL
LIN {X 0,Y 367.417,Z 477.771,A -85,B 0,C 180,E1 -12688.904,E2 -12688.904} C_VEL
LIN {X 0,Y 367.457,Z 478.139,A -85,B 0,C 180,E1 -12690,E2 -12690} C_VEL
LIN {X 0,Y 367.403,Z 478.119,A -85,B 0,C 180,E1 -12691.096,E2 -12691.096} C_VEL
LIN {X 0,Y 367.358,Z 477.716,A -85,B 0,C 180,E1 -12692.193,E2 -12692.193} C_VEL
LIN {X 0,Y 367.377,Z 476.892,A -85,B 0,C 180,E1 -12693.29,E2 -12693.29} C_VEL
LIN {X 0,Y 367.437,Z 475.652,A -85,B 0,C 180,E1 -12694.388,E2 -12694.388} C_VEL
LIN {X 0,Y 367.505,Z 473.001,A -85,B 0,C 180,E1 -12696.052,E2 -12696.052} C_VEL
LIN {X 0,Y 367.754,Z 469.402,A -85,B 0,C 180,E1 -12697.688,E2 -12697.688} C_VEL
LIN {X 0,Y 368.22,Z 464.677,A -85,B 0,C 180,E1 -12699.337,E2 -12699.337} C_VEL
LIN {X 0,Y 368.961,Z 457.595,A -85,B 0,C 180,E1 -12701.259,E2 -12701.259} C_VEL
LIN {X 0,Y 369.937,Z 449.923,A -85,B 0,C 180,E1 -12702.899,E2 -12702.899} C_VEL
LIN {X 0,Y 371.063,Z 440.645,A -85,B 0,C 180,E1 -12704.481,E2 -12704.481} C_VEL
LIN {X 0,Y 372.067,Z 430.83,A -85,B 0,C 180,E1 -12705.84,E2 -12705.84} C_VEL
LIN {X 0,Y 373.284,Z 420.662,A -85,B 0,C 180,E1 -12706.967,E2 -12706.967} C_VEL
LIN {X 0,Y 374.474,Z 408.356,A -85,B 0,C 180,E1 -12708.039,E2 -12708.039} C_VEL
LIN {X 0,Y 375.588,Z 396.306,A -85,B 0,C 180,E1 -12708.831,E2 -12708.831} C_VEL
LIN {X 0,Y 376.416,Z 383.917,A -85,B 0,C 180,E1 -12709.425,E2 -12709.425} C_VEL
LIN {X 0,Y 377.005,Z 370.593,A -85,B 0,C 180,E1 -12709.83,E2 -12709.83} C_VEL
LIN {X 0,Y 378.21,Z 298.007,A -85,B 0,C 180,E1 -12711.231,E2 -12711.231} C_VEL
LIN {X 0,Y 373.758,Z 273.428,A -85,B 0,C 180,E1 -12712.031,E2 -12712.031} C_VEL
LIN {X 0,Y 372.164,Z 265.318,A -85,B 0,C 180,E1 -12712.335,E2 -12712.335} C_VEL
LIN {X 0,Y 373.227,Z 254.283,A -85,B 0,C 180,E1 -12714.857,E2 -12714.857} C_VEL
LIN {X 0,Y 371.507,Z 244.912,A -85,B 0,C 180,E1 -12717.236,E2 -12717.236} C_VEL
LIN {X 0,Y 368.931,Z 233.526,A -85,B 0,C 180,E1 -12720.28,E2 -12720.28} C_VEL
LIN {X 0,Y 368.898,Z 233.533,A -85,B 0,C 180,E1 -12723.538,E2 -12723.538} C_VEL
LIN {X 0,Y 368.902,Z 233.533,A -85,B 0,C 180,E1 -12726.856,E2 -12726.856} C_VEL
LIN {X 0,Y 368.91,Z 233.531,A -85,B 0,C 180,E1 -12730.37,E2 -12730.37} C_VEL
LIN {X 0,Y 368.883,Z 233.538,A -85,B 0,C 180,E1 -12733.616,E2 -12733.616} C_VEL
LIN {X 0,Y 368.886,Z 233.534,A -85,B 0,C 180,E1 -12736.696,E2 -12736.696} C_VEL
LIN {X 0,Y 368.884,Z 233.537,A -85,B 0,C 180,E1 -12739.648,E2 -12739.648} C_VEL
LIN {X 0,Y 368.9,Z 233.529,A -85,B 0,C 180,E1 -12743.145,E2 -12743.145} C_VEL
LIN {X 0,Y 368.897,Z 233.526,A -85,B 0,C 180,E1 -12746.462,E2 -12746.462} C_VEL
LIN {X 0,Y 368.93,Z 233.529,A -85,B 0,C 180,E1 -12749.047,E2 -12749.047} C_VEL
LIN {X 0,Y 368.899,Z 233.531,A -85,B 0,C 180,E1 -12752.791,E2 -12752.791} C_VEL
LIN {X 0,Y 368.929,Z 233.528,A -85,B 0,C 180,E1 -12756.119,E2 -12756.119} C_VEL
LIN {X 0,Y 368.937,Z 233.527,A -85,B 0,C 180,E1 -12759.947,E2 -12759.947} C_VEL
LIN {X 0,Y 368.969,Z 233.519,A -85,B 0,C 180,E1 -12763.398,E2 -12763.398} C_VEL
LIN {X 0,Y 369.059,Z 233.511,A -85,B 0,C 180,E1 -12766.79,E2 -12766.79} C_VEL
LIN {X 0,Y 369.068,Z 233.51,A -85,B 0,C 180,E1 -12770.132,E2 -12770.132} C_VEL
LIN {X 0,Y 369.164,Z 233.492,A -85,B 0,C 180,E1 -12772.342,E2 -12772.342} C_VEL
LIN {X 0,Y 369.142,Z 233.498,A -85,B 0,C 180,E1 -12774.538,E2 -12774.538} C_VEL
LIN {X 0,Y 369.309,Z 233.474,A -85,B 0,C 180,E1 -12777.819,E2 -12777.819} C_VEL
LIN {X 0,Y 369.456,Z 233.462,A -85,B 0,C 180,E1 -12780,E2 -12780} C_VEL
LIN {X 0,Y 369.315,Z 233.474,A -85,B 0,C 180,E1 -12782.181,E2 -12782.181} C_VEL
LIN {X 0,Y 369.175,Z 233.496,A -85,B 0,C 180,E1 -12786.559,E2 -12786.559} C_VEL
LIN {X 0,Y 369.064,Z 233.512,A -85,B 0,C 180,E1 -12789.868,E2 -12789.868} C_VEL
LIN {X 0,Y 369.038,Z 233.511,A -85,B 0,C 180,E1 -12793.772,E2 -12793.772} C_VEL
LIN {X 0,Y 368.992,Z 233.514,A -85,B 0,C 180,E1 -12797.743,E2 -12797.743} C_VEL
LIN {X 0,Y 368.93,Z 233.529,A -85,B 0,C 180,E1 -12801.22,E2 -12801.22} C_VEL
LIN {X 0,Y 368.958,Z 233.523,A -85,B 0,C 180,E1 -12804.776,E2 -12804.776} C_VEL
LIN {X 0,Y 368.964,Z 233.52,A -85,B 0,C 180,E1 -12807.204,E2 -12807.204} C_VEL
LIN {X 0,Y 368.931,Z 233.525,A -85,B 0,C 180,E1 -12810.954,E2 -12810.954} C_VEL
LIN {X 0,Y 368.93,Z 233.529,A -85,B 0,C 180,E1 -12815.002,E2 -12815.002} C_VEL
LIN {X 0,Y 368.908,Z 233.53,A -85,B 0,C 180,E1 -12818.64,E2 -12818.64} C_VEL
LIN {X 0,Y 368.882,Z 233.535,A -85,B 0,C 180,E1 -12822.009,E2 -12822.009} C_VEL
LIN {X 0,Y 368.927,Z 233.534,A -85,B 0,C 180,E1 -12825.183,E2 -12825.183} C_VEL
LIN {X 0,Y 368.873,Z 233.54,A -85,B 0,C 180,E1 -12828.176,E2 -12828.176} C_VEL
LIN {X 0,Y 368.88,Z 233.541,A -85,B 0,C 180,E1 -12831.366,E2 -12831.366} C_VEL
LIN {X 0,Y 368.938,Z 233.533,A -85,B 0,C 180,E1 -12835.147,E2 -12835.147} C_VEL
LIN {X 0,Y 368.927,Z 233.62,A -85,B 0,C 180,E1 -12838.032,E2 -12838.032} C_VEL
LIN {X 0,Y 371.4,Z 244.822,A -85,B 0,C 180,E1 -12841.149,E2 -12841.149} C_VEL
LIN {X 0,Y 371.833,Z 247.079,A -85,B 0,C 180,E1 -12841.715,E2 -12841.715} C_VEL
LIN {X 0,Y 374.675,Z 255.29,A -85,B 0,C 180,E1 -12842.085,E2 -12842.085} C_VEL
LIN {X 0,Y 378.665,Z 272.901,A -85,B 0,C 180,E1 -12842.717,E2 -12842.717} C_VEL
LIN {X 0,Y 377.168,Z 354.126,A -85,B 0,C 180,E1 -12844.29,E2 -12844.29} C_VEL
LIN {X 0,Y 376.571,Z 367.57,A -85,B 0,C 180,E1 -12844.765,E2 -12844.765} C_VEL
LIN {X 0,Y 375.842,Z 379.85,A -85,B 0,C 180,E1 -12845.414,E2 -12845.414} C_VEL
LIN {X 0,Y 374.872,Z 391.361,A -85,B 0,C 180,E1 -12846.229,E2 -12846.229} C_VEL
LIN {X 0,Y 373.828,Z 402.469,A -85,B 0,C 180,E1 -12847.255,E2 -12847.255} C_VEL
LIN {X 0,Y 372.479,Z 413.7,A -85,B 0,C 180,E1 -12848.557,E2 -12848.557} C_VEL
LIN {X 0,Y 371.58,Z 422.308,A -85,B 0,C 180,E1 -12849.807,E2 -12849.807} C_VEL
LIN {X 0,Y 370.586,Z 430.206,A -85,B 0,C 180,E1 -12851.192,E2 -12851.192} C_VEL
LIN {X 0,Y 369.624,Z 437.881,A -85,B 0,C 180,E1 -12852.859,E2 -12852.859} C_VEL
LIN {X 0,Y 368.859,Z 444.024,A -85,B 0,C 180,E1 -12854.529,E2 -12854.529} C_VEL
LIN {X 0,Y 368.305,Z 448.875,A -85,B 0,C 180,E1 -12856.2,E2 -12856.2} C_VEL
LIN {X 0,Y 367.882,Z 452.587,A -85,B 0,C 180,E1 -12857.869,E2 -12857.869} C_VEL
LIN {X 0,Y 367.651,Z 454.496,A -85,B 0,C 180,E1 -12858.98,E2 -12858.98} C_VEL
LIN {X 0,Y 367.478,Z 455.961,A -85,B 0,C 180,E1 -12860.089,E2 -12860.089} C_VEL
LIN {X 0,Y 367.407,Z 457.616,A -85,B 0,C 180,E1 -12862.305,E2 -12862.305} C_VEL
LIN {X 0,Y 367.482,Z 457.811,A -85,B 0,C 180,E1 -12863.985,E2 -12863.985} C_VEL
LIN {X 0,Y 367.428,Z 457.129,A -85,B 0,C 180,E1 -12865.612,E2 -12865.612} C_VEL
LIN {X 0,Y 367.471,Z 454.823,A -85,B 0,C 180,E1 -12867.808,E2 -12867.808} C_VEL
LIN {X 0,Y 367.638,Z 451.976,A -85,B 0,C 180,E1 -12869.452,E2 -12869.452} C_VEL
LIN {X 0,Y 367.844,Z 448.119,A -85,B 0,C 180,E1 -12871.095,E2 -12871.095} C_VEL
LIN {X 0,Y 368.276,Z 443.138,A -85,B 0,C 180,E1 -12872.735,E2 -12872.735} C_VEL
LIN {X 0,Y 368.784,Z 436.891,A -85,B 0,C 180,E1 -12874.372,E2 -12874.372} C_VEL
LIN {X 0,Y 369.528,Z 429.069,A -85,B 0,C 180,E1 -12876.004,E2 -12876.004} C_VEL
LIN {X 0,Y 370.348,Z 421.099,A -85,B 0,C 180,E1 -12877.359,E2 -12877.359} C_VEL
LIN {X 0,Y 371.268,Z 411.387,A -85,B 0,C 180,E1 -12878.71,E2 -12878.71} C_VEL
LIN {X 0,Y 372.213,Z 400.56,A -85,B 0,C 180,E1 -12879.921,E2 -12879.921} C_VEL
LIN {X 0,Y 373.126,Z 388.216,A -85,B 0,C 180,E1 -12880.994,E2 -12880.994} C_VEL
LIN {X 0,Y 373.884,Z 376.109,A -85,B 0,C 180,E1 -12881.796,E2 -12881.796} C_VEL
